REGION Network 60: STATUS - UNIT 01 - ST2
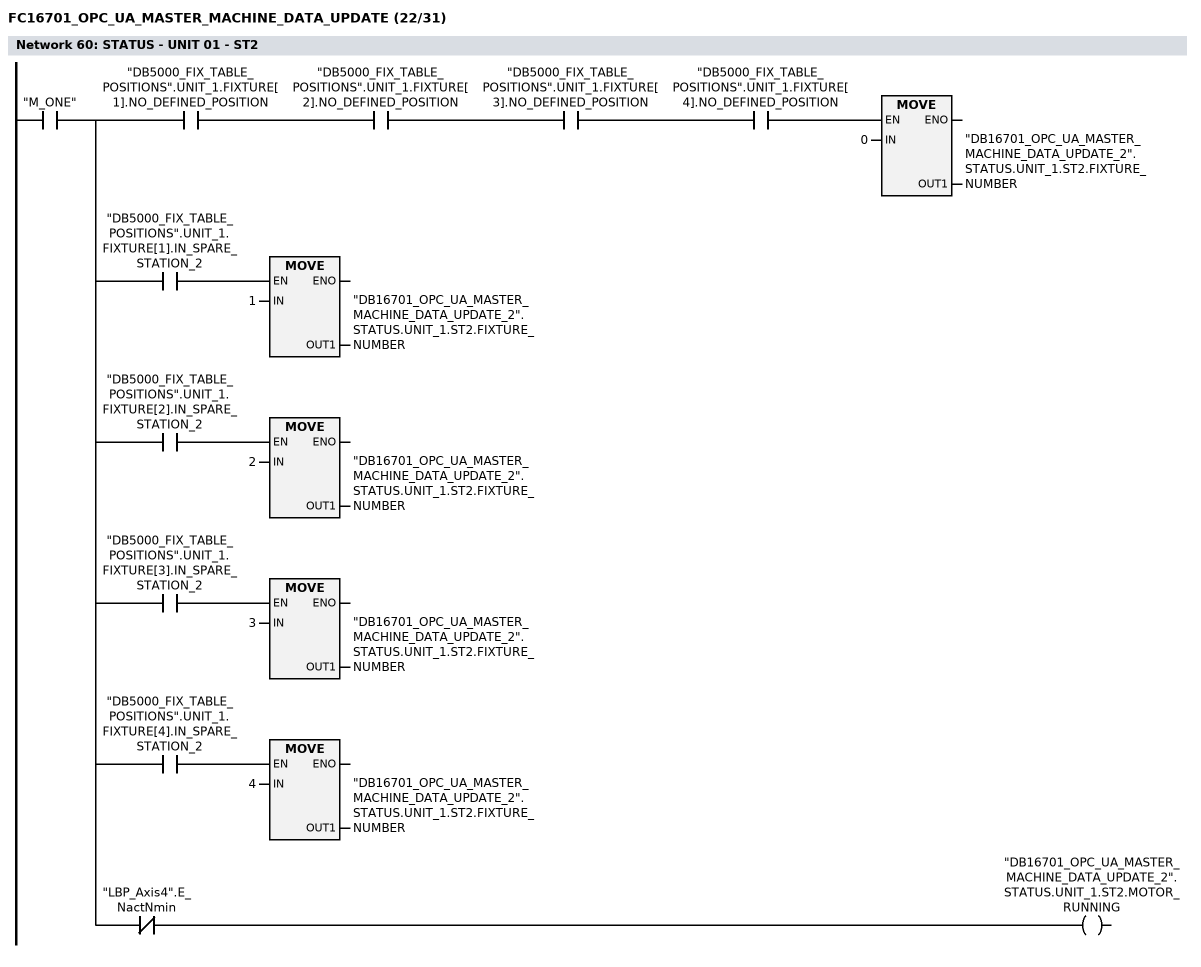
   RUNG wire#powerrail
      Contact( "M_ONE" )
      wire#w1
      Contact( "DB5000_FIX_TABLE_POSITIONS".UNIT_1.FIXTURE[1].NO_DEFINED_POSITION )
      Contact( "DB5000_FIX_TABLE_POSITIONS".UNIT_1.FIXTURE[2].NO_DEFINED_POSITION )
      Contact( "DB5000_FIX_TABLE_POSITIONS".UNIT_1.FIXTURE[3].NO_DEFINED_POSITION )
      Contact( "DB5000_FIX_TABLE_POSITIONS".UNIT_1.FIXTURE[4].NO_DEFINED_POSITION )
      Move(in := 0, out1 => "DB16701_OPC_UA_MASTER_MACHINE_DATA_UPDATE_2".STATUS.UNIT_1.ST2.FIXTURE_NUMBER)
   END_RUNG
   RUNG wire#w1
      Contact( "DB5000_FIX_TABLE_POSITIONS".UNIT_1.FIXTURE[1].IN_SPARE_STATION_2 )
      Move(in := 1, out1 => "DB16701_OPC_UA_MASTER_MACHINE_DATA_UPDATE_2".STATUS.UNIT_1.ST2.FIXTURE_NUMBER)
   END_RUNG
   RUNG wire#w1
      Contact( "DB5000_FIX_TABLE_POSITIONS".UNIT_1.FIXTURE[2].IN_SPARE_STATION_2 )
      Move(in := 2, out1 => "DB16701_OPC_UA_MASTER_MACHINE_DATA_UPDATE_2".STATUS.UNIT_1.ST2.FIXTURE_NUMBER)
   END_RUNG
   RUNG wire#w1
      Contact( "DB5000_FIX_TABLE_POSITIONS".UNIT_1.FIXTURE[3].IN_SPARE_STATION_2 )
      Move(in := 3, out1 => "DB16701_OPC_UA_MASTER_MACHINE_DATA_UPDATE_2".STATUS.UNIT_1.ST2.FIXTURE_NUMBER)
   END_RUNG
   RUNG wire#w1
      Contact( "DB5000_FIX_TABLE_POSITIONS".UNIT_1.FIXTURE[4].IN_SPARE_STATION_2 )
      Move(in := 4, out1 => "DB16701_OPC_UA_MASTER_MACHINE_DATA_UPDATE_2".STATUS.UNIT_1.ST2.FIXTURE_NUMBER)
   END_RUNG
   RUNG wire#w1
      I_Contact( "LBP_Axis4".E_NactNmin )
      Coil( "DB16701_OPC_UA_MASTER_MACHINE_DATA_UPDATE_2".STATUS.UNIT_1.ST2.MOTOR_RUNNING )
   END_RUNG
   // the same network as SCL:
   IF "M_ONE" AND "DB5000_FIX_TABLE_POSITIONS".UNIT_1.FIXTURE[1].NO_DEFINED_POSITION AND "DB5000_FIX_TABLE_POSITIONS".UNIT_1.FIXTURE[2].NO_DEFINED_POSITION AND "DB5000_FIX_TABLE_POSITIONS".UNIT_1.FIXTURE[3].NO_DEFINED_POSITION AND "DB5000_FIX_TABLE_POSITIONS".UNIT_1.FIXTURE[4].NO_DEFINED_POSITION THEN
       "DB16701_OPC_UA_MASTER_MACHINE_DATA_UPDATE_2".STATUS.UNIT_1.ST2.FIXTURE_NUMBER := 0;
   END_IF;
   IF "M_ONE" AND "DB5000_FIX_TABLE_POSITIONS".UNIT_1.FIXTURE[1].IN_SPARE_STATION_2 THEN
       "DB16701_OPC_UA_MASTER_MACHINE_DATA_UPDATE_2".STATUS.UNIT_1.ST2.FIXTURE_NUMBER := 1;
   END_IF;
   IF "M_ONE" AND "DB5000_FIX_TABLE_POSITIONS".UNIT_1.FIXTURE[2].IN_SPARE_STATION_2 THEN
       "DB16701_OPC_UA_MASTER_MACHINE_DATA_UPDATE_2".STATUS.UNIT_1.ST2.FIXTURE_NUMBER := 2;
   END_IF;
   IF "M_ONE" AND "DB5000_FIX_TABLE_POSITIONS".UNIT_1.FIXTURE[3].IN_SPARE_STATION_2 THEN
       "DB16701_OPC_UA_MASTER_MACHINE_DATA_UPDATE_2".STATUS.UNIT_1.ST2.FIXTURE_NUMBER := 3;
   END_IF;
   IF "M_ONE" AND "DB5000_FIX_TABLE_POSITIONS".UNIT_1.FIXTURE[4].IN_SPARE_STATION_2 THEN
       "DB16701_OPC_UA_MASTER_MACHINE_DATA_UPDATE_2".STATUS.UNIT_1.ST2.FIXTURE_NUMBER := 4;
   END_IF;
   "DB16701_OPC_UA_MASTER_MACHINE_DATA_UPDATE_2".STATUS.UNIT_1.ST2.MOTOR_RUNNING := "M_ONE" AND NOT "LBP_Axis4".E_NactNmin;
END_REGION

REGION Network 61: STATUS - UNIT 01 - ST3
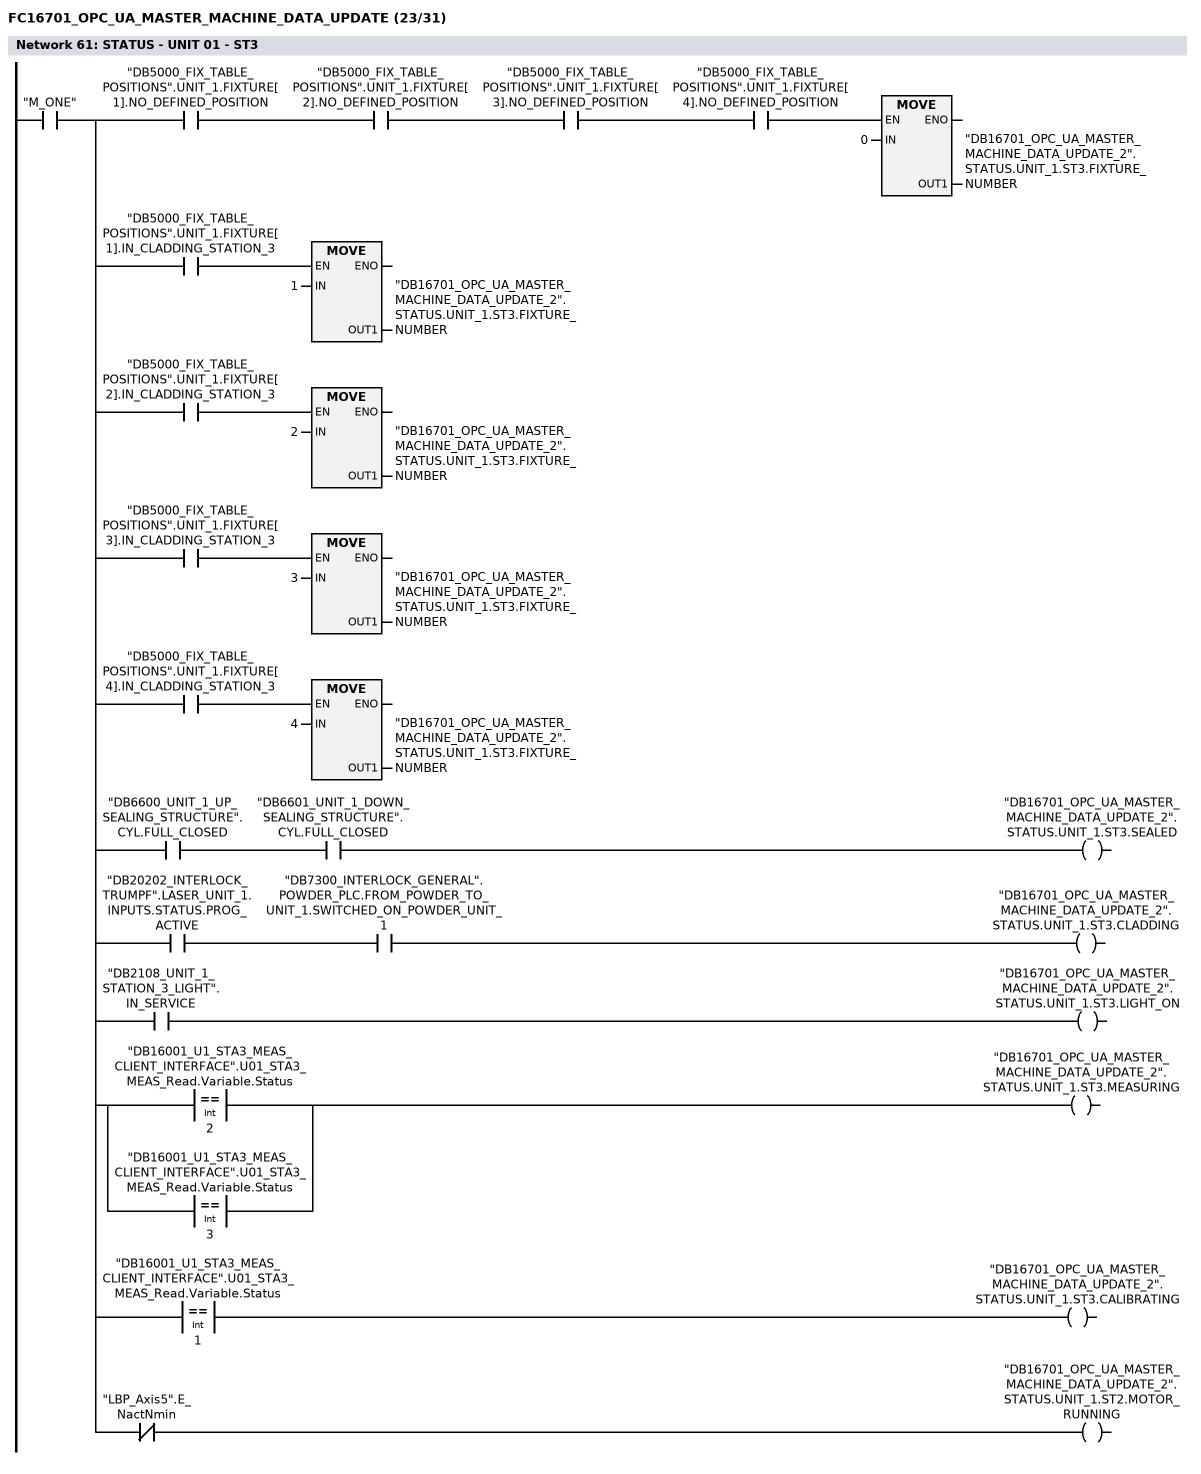
   RUNG wire#powerrail
      Contact( "M_ONE" )
      wire#w1
      Contact( "DB5000_FIX_TABLE_POSITIONS".UNIT_1.FIXTURE[1].NO_DEFINED_POSITION )
      Contact( "DB5000_FIX_TABLE_POSITIONS".UNIT_1.FIXTURE[2].NO_DEFINED_POSITION )
      Contact( "DB5000_FIX_TABLE_POSITIONS".UNIT_1.FIXTURE[3].NO_DEFINED_POSITION )
      Contact( "DB5000_FIX_TABLE_POSITIONS".UNIT_1.FIXTURE[4].NO_DEFINED_POSITION )
      Move(in := 0, out1 => "DB16701_OPC_UA_MASTER_MACHINE_DATA_UPDATE_2".STATUS.UNIT_1.ST3.FIXTURE_NUMBER)
   END_RUNG
   RUNG wire#w1
      Contact( "DB5000_FIX_TABLE_POSITIONS".UNIT_1.FIXTURE[1].IN_CLADDING_STATION_3 )
      Move(in := 1, out1 => "DB16701_OPC_UA_MASTER_MACHINE_DATA_UPDATE_2".STATUS.UNIT_1.ST3.FIXTURE_NUMBER)
   END_RUNG
   RUNG wire#w1
      Contact( "DB5000_FIX_TABLE_POSITIONS".UNIT_1.FIXTURE[2].IN_CLADDING_STATION_3 )
      Move(in := 2, out1 => "DB16701_OPC_UA_MASTER_MACHINE_DATA_UPDATE_2".STATUS.UNIT_1.ST3.FIXTURE_NUMBER)
   END_RUNG
   RUNG wire#w1
      Contact( "DB5000_FIX_TABLE_POSITIONS".UNIT_1.FIXTURE[3].IN_CLADDING_STATION_3 )
      Move(in := 3, out1 => "DB16701_OPC_UA_MASTER_MACHINE_DATA_UPDATE_2".STATUS.UNIT_1.ST3.FIXTURE_NUMBER)
   END_RUNG
   RUNG wire#w1
      Contact( "DB5000_FIX_TABLE_POSITIONS".UNIT_1.FIXTURE[4].IN_CLADDING_STATION_3 )
      Move(in := 4, out1 => "DB16701_OPC_UA_MASTER_MACHINE_DATA_UPDATE_2".STATUS.UNIT_1.ST3.FIXTURE_NUMBER)
   END_RUNG
   RUNG wire#w1
      Contact( "DB6600_UNIT_1_UP_SEALING_STRUCTURE".CYL.FULL_CLOSED )
      Contact( "DB6601_UNIT_1_DOWN_SEALING_STRUCTURE".CYL.FULL_CLOSED )
      Coil( "DB16701_OPC_UA_MASTER_MACHINE_DATA_UPDATE_2".STATUS.UNIT_1.ST3.SEALED )
   END_RUNG
   RUNG wire#w1
      Contact( "DB20202_INTERLOCK_TRUMPF".LASER_UNIT_1.INPUTS.STATUS.PROG_ACTIVE )
      Contact( "DB7300_INTERLOCK_GENERAL".POWDER_PLC.FROM_POWDER_TO_UNIT_1.SWITCHED_ON_POWDER_UNIT_1 )
      Coil( "DB16701_OPC_UA_MASTER_MACHINE_DATA_UPDATE_2".STATUS.UNIT_1.ST3.CLADDING )
   END_RUNG
   RUNG wire#w1
      Contact( "DB2108_UNIT_1_STATION_3_LIGHT".IN_SERVICE )
      Coil( "DB16701_OPC_UA_MASTER_MACHINE_DATA_UPDATE_2".STATUS.UNIT_1.ST3.LIGHT_ON )
   END_RUNG
   RUNG wire#w1
      { S7_Templates := "SrcType := Int" } EQ_Contact(in1 := "DB16001_U1_STA3_MEAS_CLIENT_INTERFACE".U01_STA3_MEAS_Read.Variable.Status, in2 := 2)
      wire#w2
      Coil( "DB16701_OPC_UA_MASTER_MACHINE_DATA_UPDATE_2".STATUS.UNIT_1.ST3.MEASURING )
   END_RUNG
   RUNG wire#w1
      { S7_Templates := "SrcType := Int" } EQ_Contact(in1 := "DB16001_U1_STA3_MEAS_CLIENT_INTERFACE".U01_STA3_MEAS_Read.Variable.Status, in2 := 3)
   END_RUNG wire#w2
   RUNG wire#w1
      { S7_Templates := "SrcType := Int" } EQ_Contact(in1 := "DB16001_U1_STA3_MEAS_CLIENT_INTERFACE".U01_STA3_MEAS_Read.Variable.Status, in2 := 1)
      Coil( "DB16701_OPC_UA_MASTER_MACHINE_DATA_UPDATE_2".STATUS.UNIT_1.ST3.CALIBRATING )
   END_RUNG
   RUNG wire#w1
      I_Contact( "LBP_Axis5".E_NactNmin )
      Coil( "DB16701_OPC_UA_MASTER_MACHINE_DATA_UPDATE_2".STATUS.UNIT_1.ST2.MOTOR_RUNNING )
   END_RUNG
   // the same network as SCL:
   IF "M_ONE" AND "DB5000_FIX_TABLE_POSITIONS".UNIT_1.FIXTURE[1].NO_DEFINED_POSITION AND "DB5000_FIX_TABLE_POSITIONS".UNIT_1.FIXTURE[2].NO_DEFINED_POSITION AND "DB5000_FIX_TABLE_POSITIONS".UNIT_1.FIXTURE[3].NO_DEFINED_POSITION AND "DB5000_FIX_TABLE_POSITIONS".UNIT_1.FIXTURE[4].NO_DEFINED_POSITION THEN
       "DB16701_OPC_UA_MASTER_MACHINE_DATA_UPDATE_2".STATUS.UNIT_1.ST3.FIXTURE_NUMBER := 0;
   END_IF;
   IF "M_ONE" AND "DB5000_FIX_TABLE_POSITIONS".UNIT_1.FIXTURE[1].IN_CLADDING_STATION_3 THEN
       "DB16701_OPC_UA_MASTER_MACHINE_DATA_UPDATE_2".STATUS.UNIT_1.ST3.FIXTURE_NUMBER := 1;
   END_IF;
   IF "M_ONE" AND "DB5000_FIX_TABLE_POSITIONS".UNIT_1.FIXTURE[2].IN_CLADDING_STATION_3 THEN
       "DB16701_OPC_UA_MASTER_MACHINE_DATA_UPDATE_2".STATUS.UNIT_1.ST3.FIXTURE_NUMBER := 2;
   END_IF;
   IF "M_ONE" AND "DB5000_FIX_TABLE_POSITIONS".UNIT_1.FIXTURE[3].IN_CLADDING_STATION_3 THEN
       "DB16701_OPC_UA_MASTER_MACHINE_DATA_UPDATE_2".STATUS.UNIT_1.ST3.FIXTURE_NUMBER := 3;
   END_IF;
   IF "M_ONE" AND "DB5000_FIX_TABLE_POSITIONS".UNIT_1.FIXTURE[4].IN_CLADDING_STATION_3 THEN
       "DB16701_OPC_UA_MASTER_MACHINE_DATA_UPDATE_2".STATUS.UNIT_1.ST3.FIXTURE_NUMBER := 4;
   END_IF;
   "DB16701_OPC_UA_MASTER_MACHINE_DATA_UPDATE_2".STATUS.UNIT_1.ST3.SEALED := "M_ONE" AND "DB6600_UNIT_1_UP_SEALING_STRUCTURE".CYL.FULL_CLOSED AND "DB6601_UNIT_1_DOWN_SEALING_STRUCTURE".CYL.FULL_CLOSED;
   "DB16701_OPC_UA_MASTER_MACHINE_DATA_UPDATE_2".STATUS.UNIT_1.ST3.CLADDING := "M_ONE" AND "DB20202_INTERLOCK_TRUMPF".LASER_UNIT_1.INPUTS.STATUS.PROG_ACTIVE AND "DB7300_INTERLOCK_GENERAL".POWDER_PLC.FROM_POWDER_TO_UNIT_1.SWITCHED_ON_POWDER_UNIT_1;
   "DB16701_OPC_UA_MASTER_MACHINE_DATA_UPDATE_2".STATUS.UNIT_1.ST3.LIGHT_ON := "M_ONE" AND "DB2108_UNIT_1_STATION_3_LIGHT".IN_SERVICE;
   "DB16701_OPC_UA_MASTER_MACHINE_DATA_UPDATE_2".STATUS.UNIT_1.ST3.MEASURING := "M_ONE" AND (("DB16001_U1_STA3_MEAS_CLIENT_INTERFACE".U01_STA3_MEAS_Read.Variable.Status = 2) OR ("DB16001_U1_STA3_MEAS_CLIENT_INTERFACE".U01_STA3_MEAS_Read.Variable.Status = 3));
   "DB16701_OPC_UA_MASTER_MACHINE_DATA_UPDATE_2".STATUS.UNIT_1.ST3.CALIBRATING := "M_ONE" AND ("DB16001_U1_STA3_MEAS_CLIENT_INTERFACE".U01_STA3_MEAS_Read.Variable.Status = 1);
   "DB16701_OPC_UA_MASTER_MACHINE_DATA_UPDATE_2".STATUS.UNIT_1.ST2.MOTOR_RUNNING := "M_ONE" AND NOT "LBP_Axis5".E_NactNmin;
END_REGION

REGION Network 62: STATUS - UNIT 01 - ST4
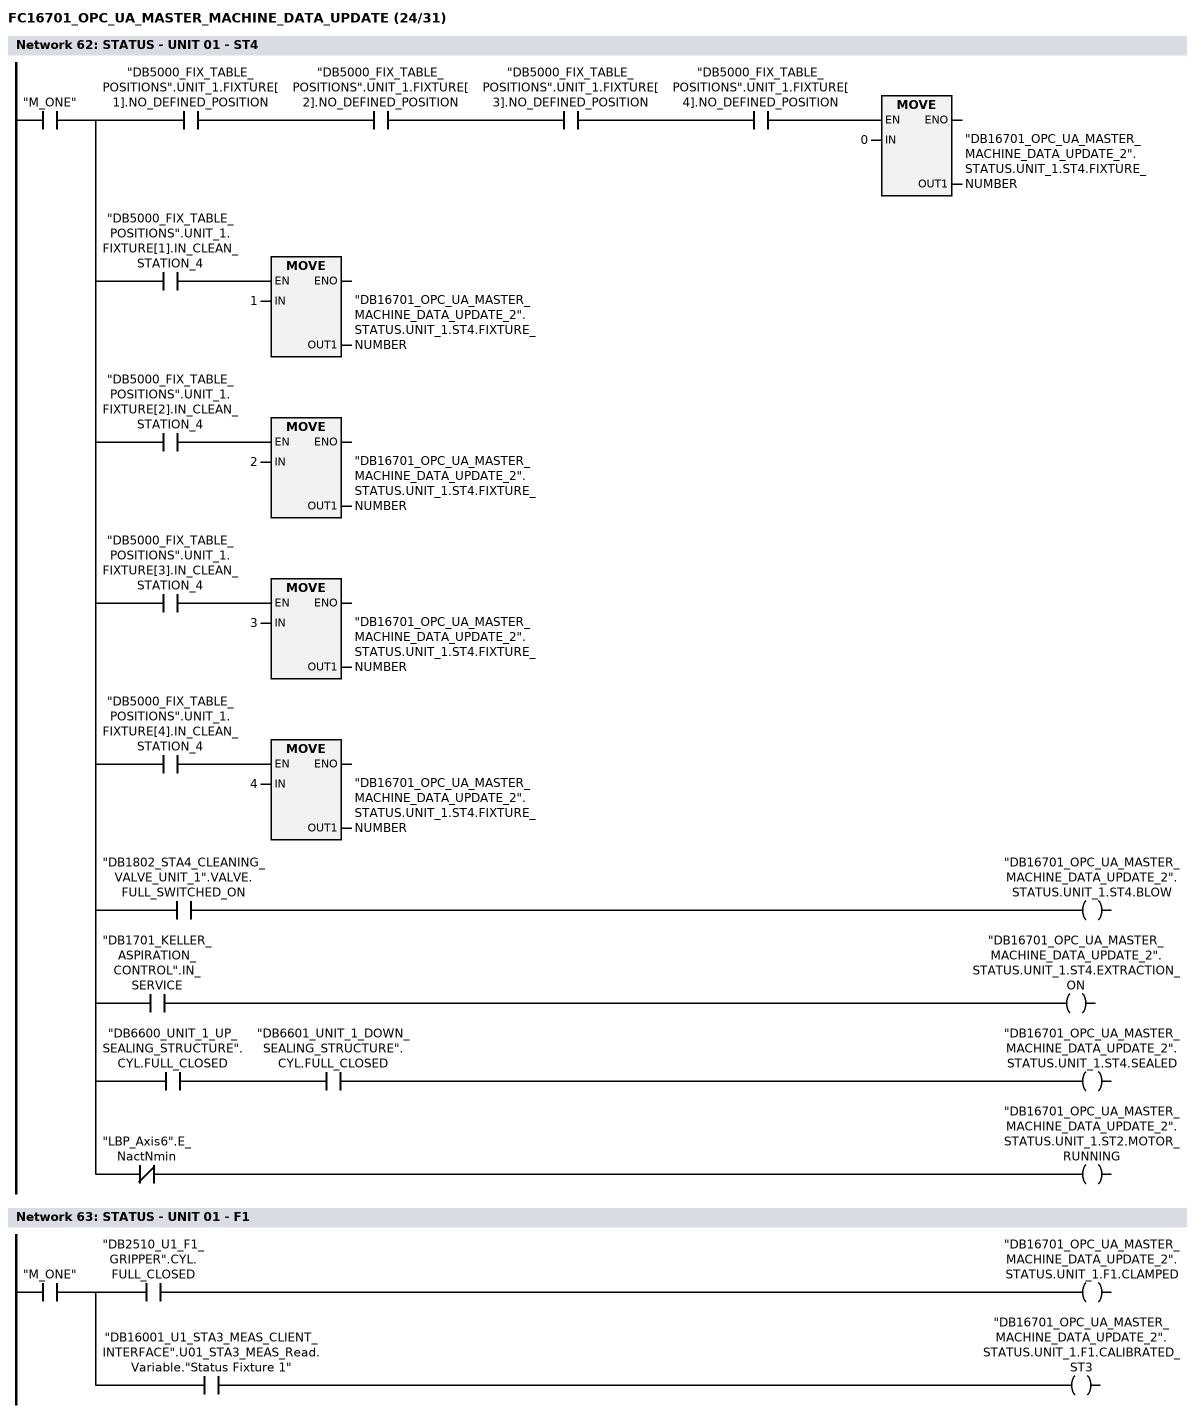
   RUNG wire#powerrail
      Contact( "M_ONE" )
      wire#w1
      Contact( "DB5000_FIX_TABLE_POSITIONS".UNIT_1.FIXTURE[1].NO_DEFINED_POSITION )
      Contact( "DB5000_FIX_TABLE_POSITIONS".UNIT_1.FIXTURE[2].NO_DEFINED_POSITION )
      Contact( "DB5000_FIX_TABLE_POSITIONS".UNIT_1.FIXTURE[3].NO_DEFINED_POSITION )
      Contact( "DB5000_FIX_TABLE_POSITIONS".UNIT_1.FIXTURE[4].NO_DEFINED_POSITION )
      Move(in := 0, out1 => "DB16701_OPC_UA_MASTER_MACHINE_DATA_UPDATE_2".STATUS.UNIT_1.ST4.FIXTURE_NUMBER)
   END_RUNG
   RUNG wire#w1
      Contact( "DB5000_FIX_TABLE_POSITIONS".UNIT_1.FIXTURE[1].IN_CLEAN_STATION_4 )
      Move(in := 1, out1 => "DB16701_OPC_UA_MASTER_MACHINE_DATA_UPDATE_2".STATUS.UNIT_1.ST4.FIXTURE_NUMBER)
   END_RUNG
   RUNG wire#w1
      Contact( "DB5000_FIX_TABLE_POSITIONS".UNIT_1.FIXTURE[2].IN_CLEAN_STATION_4 )
      Move(in := 2, out1 => "DB16701_OPC_UA_MASTER_MACHINE_DATA_UPDATE_2".STATUS.UNIT_1.ST4.FIXTURE_NUMBER)
   END_RUNG
   RUNG wire#w1
      Contact( "DB5000_FIX_TABLE_POSITIONS".UNIT_1.FIXTURE[3].IN_CLEAN_STATION_4 )
      Move(in := 3, out1 => "DB16701_OPC_UA_MASTER_MACHINE_DATA_UPDATE_2".STATUS.UNIT_1.ST4.FIXTURE_NUMBER)
   END_RUNG
   RUNG wire#w1
      Contact( "DB5000_FIX_TABLE_POSITIONS".UNIT_1.FIXTURE[4].IN_CLEAN_STATION_4 )
      Move(in := 4, out1 => "DB16701_OPC_UA_MASTER_MACHINE_DATA_UPDATE_2".STATUS.UNIT_1.ST4.FIXTURE_NUMBER)
   END_RUNG
   RUNG wire#w1
      Contact( "DB1802_STA4_CLEANING_VALVE_UNIT_1".VALVE.FULL_SWITCHED_ON )
      Coil( "DB16701_OPC_UA_MASTER_MACHINE_DATA_UPDATE_2".STATUS.UNIT_1.ST4.BLOW )
   END_RUNG
   RUNG wire#w1
      Contact( "DB1701_KELLER_ASPIRATION_CONTROL".IN_SERVICE )
      Coil( "DB16701_OPC_UA_MASTER_MACHINE_DATA_UPDATE_2".STATUS.UNIT_1.ST4.EXTRACTION_ON )
   END_RUNG
   RUNG wire#w1
      Contact( "DB6600_UNIT_1_UP_SEALING_STRUCTURE".CYL.FULL_CLOSED )
      Contact( "DB6601_UNIT_1_DOWN_SEALING_STRUCTURE".CYL.FULL_CLOSED )
      Coil( "DB16701_OPC_UA_MASTER_MACHINE_DATA_UPDATE_2".STATUS.UNIT_1.ST4.SEALED )
   END_RUNG
   RUNG wire#w1
      I_Contact( "LBP_Axis6".E_NactNmin )
      Coil( "DB16701_OPC_UA_MASTER_MACHINE_DATA_UPDATE_2".STATUS.UNIT_1.ST2.MOTOR_RUNNING )
   END_RUNG
   // the same network as SCL:
   IF "M_ONE" AND "DB5000_FIX_TABLE_POSITIONS".UNIT_1.FIXTURE[1].NO_DEFINED_POSITION AND "DB5000_FIX_TABLE_POSITIONS".UNIT_1.FIXTURE[2].NO_DEFINED_POSITION AND "DB5000_FIX_TABLE_POSITIONS".UNIT_1.FIXTURE[3].NO_DEFINED_POSITION AND "DB5000_FIX_TABLE_POSITIONS".UNIT_1.FIXTURE[4].NO_DEFINED_POSITION THEN
       "DB16701_OPC_UA_MASTER_MACHINE_DATA_UPDATE_2".STATUS.UNIT_1.ST4.FIXTURE_NUMBER := 0;
   END_IF;
   IF "M_ONE" AND "DB5000_FIX_TABLE_POSITIONS".UNIT_1.FIXTURE[1].IN_CLEAN_STATION_4 THEN
       "DB16701_OPC_UA_MASTER_MACHINE_DATA_UPDATE_2".STATUS.UNIT_1.ST4.FIXTURE_NUMBER := 1;
   END_IF;
   IF "M_ONE" AND "DB5000_FIX_TABLE_POSITIONS".UNIT_1.FIXTURE[2].IN_CLEAN_STATION_4 THEN
       "DB16701_OPC_UA_MASTER_MACHINE_DATA_UPDATE_2".STATUS.UNIT_1.ST4.FIXTURE_NUMBER := 2;
   END_IF;
   IF "M_ONE" AND "DB5000_FIX_TABLE_POSITIONS".UNIT_1.FIXTURE[3].IN_CLEAN_STATION_4 THEN
       "DB16701_OPC_UA_MASTER_MACHINE_DATA_UPDATE_2".STATUS.UNIT_1.ST4.FIXTURE_NUMBER := 3;
   END_IF;
   IF "M_ONE" AND "DB5000_FIX_TABLE_POSITIONS".UNIT_1.FIXTURE[4].IN_CLEAN_STATION_4 THEN
       "DB16701_OPC_UA_MASTER_MACHINE_DATA_UPDATE_2".STATUS.UNIT_1.ST4.FIXTURE_NUMBER := 4;
   END_IF;
   "DB16701_OPC_UA_MASTER_MACHINE_DATA_UPDATE_2".STATUS.UNIT_1.ST4.BLOW := "M_ONE" AND "DB1802_STA4_CLEANING_VALVE_UNIT_1".VALVE.FULL_SWITCHED_ON;
   "DB16701_OPC_UA_MASTER_MACHINE_DATA_UPDATE_2".STATUS.UNIT_1.ST4.EXTRACTION_ON := "M_ONE" AND "DB1701_KELLER_ASPIRATION_CONTROL".IN_SERVICE;
   "DB16701_OPC_UA_MASTER_MACHINE_DATA_UPDATE_2".STATUS.UNIT_1.ST4.SEALED := "M_ONE" AND "DB6600_UNIT_1_UP_SEALING_STRUCTURE".CYL.FULL_CLOSED AND "DB6601_UNIT_1_DOWN_SEALING_STRUCTURE".CYL.FULL_CLOSED;
   "DB16701_OPC_UA_MASTER_MACHINE_DATA_UPDATE_2".STATUS.UNIT_1.ST2.MOTOR_RUNNING := "M_ONE" AND NOT "LBP_Axis6".E_NactNmin;
END_REGION

REGION Network 63: STATUS - UNIT 01 - F1
   RUNG wire#powerrail
      Contact( "M_ONE" )
      wire#w1
      Contact( "DB2510_U1_F1_GRIPPER".CYL.FULL_CLOSED )
      Coil( "DB16701_OPC_UA_MASTER_MACHINE_DATA_UPDATE_2".STATUS.UNIT_1.F1.CLAMPED )
   END_RUNG
   RUNG wire#w1
      Contact( "DB16001_U1_STA3_MEAS_CLIENT_INTERFACE".U01_STA3_MEAS_Read.Variable."Status Fixture 1" )
      Coil( "DB16701_OPC_UA_MASTER_MACHINE_DATA_UPDATE_2".STATUS.UNIT_1.F1.CALIBRATED_ST3 )
   END_RUNG
   // the same network as SCL:
   "DB16701_OPC_UA_MASTER_MACHINE_DATA_UPDATE_2".STATUS.UNIT_1.F1.CLAMPED := "M_ONE" AND "DB2510_U1_F1_GRIPPER".CYL.FULL_CLOSED;
   "DB16701_OPC_UA_MASTER_MACHINE_DATA_UPDATE_2".STATUS.UNIT_1.F1.CALIBRATED_ST3 := "M_ONE" AND "DB16001_U1_STA3_MEAS_CLIENT_INTERFACE".U01_STA3_MEAS_Read.Variable."Status Fixture 1";
END_REGION

REGION Network 64: STATUS - UNIT 01 - F2
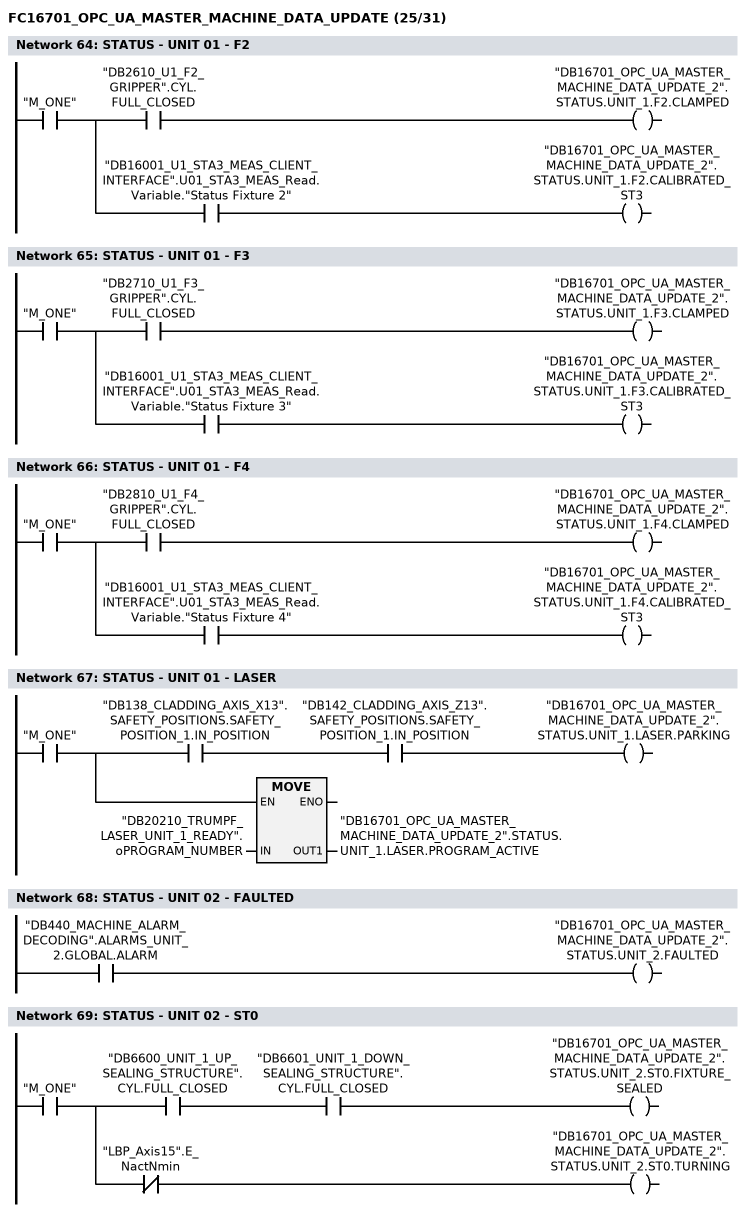
   RUNG wire#powerrail
      Contact( "M_ONE" )
      wire#w1
      Contact( "DB2610_U1_F2_GRIPPER".CYL.FULL_CLOSED )
      Coil( "DB16701_OPC_UA_MASTER_MACHINE_DATA_UPDATE_2".STATUS.UNIT_1.F2.CLAMPED )
   END_RUNG
   RUNG wire#w1
      Contact( "DB16001_U1_STA3_MEAS_CLIENT_INTERFACE".U01_STA3_MEAS_Read.Variable."Status Fixture 2" )
      Coil( "DB16701_OPC_UA_MASTER_MACHINE_DATA_UPDATE_2".STATUS.UNIT_1.F2.CALIBRATED_ST3 )
   END_RUNG
   // the same network as SCL:
   "DB16701_OPC_UA_MASTER_MACHINE_DATA_UPDATE_2".STATUS.UNIT_1.F2.CLAMPED := "M_ONE" AND "DB2610_U1_F2_GRIPPER".CYL.FULL_CLOSED;
   "DB16701_OPC_UA_MASTER_MACHINE_DATA_UPDATE_2".STATUS.UNIT_1.F2.CALIBRATED_ST3 := "M_ONE" AND "DB16001_U1_STA3_MEAS_CLIENT_INTERFACE".U01_STA3_MEAS_Read.Variable."Status Fixture 2";
END_REGION

REGION Network 65: STATUS - UNIT 01 - F3
   RUNG wire#powerrail
      Contact( "M_ONE" )
      wire#w1
      Contact( "DB2710_U1_F3_GRIPPER".CYL.FULL_CLOSED )
      Coil( "DB16701_OPC_UA_MASTER_MACHINE_DATA_UPDATE_2".STATUS.UNIT_1.F3.CLAMPED )
   END_RUNG
   RUNG wire#w1
      Contact( "DB16001_U1_STA3_MEAS_CLIENT_INTERFACE".U01_STA3_MEAS_Read.Variable."Status Fixture 3" )
      Coil( "DB16701_OPC_UA_MASTER_MACHINE_DATA_UPDATE_2".STATUS.UNIT_1.F3.CALIBRATED_ST3 )
   END_RUNG
   // the same network as SCL:
   "DB16701_OPC_UA_MASTER_MACHINE_DATA_UPDATE_2".STATUS.UNIT_1.F3.CLAMPED := "M_ONE" AND "DB2710_U1_F3_GRIPPER".CYL.FULL_CLOSED;
   "DB16701_OPC_UA_MASTER_MACHINE_DATA_UPDATE_2".STATUS.UNIT_1.F3.CALIBRATED_ST3 := "M_ONE" AND "DB16001_U1_STA3_MEAS_CLIENT_INTERFACE".U01_STA3_MEAS_Read.Variable."Status Fixture 3";
END_REGION

REGION Network 66: STATUS - UNIT 01 - F4
   RUNG wire#powerrail
      Contact( "M_ONE" )
      wire#w1
      Contact( "DB2810_U1_F4_GRIPPER".CYL.FULL_CLOSED )
      Coil( "DB16701_OPC_UA_MASTER_MACHINE_DATA_UPDATE_2".STATUS.UNIT_1.F4.CLAMPED )
   END_RUNG
   RUNG wire#w1
      Contact( "DB16001_U1_STA3_MEAS_CLIENT_INTERFACE".U01_STA3_MEAS_Read.Variable."Status Fixture 4" )
      Coil( "DB16701_OPC_UA_MASTER_MACHINE_DATA_UPDATE_2".STATUS.UNIT_1.F4.CALIBRATED_ST3 )
   END_RUNG
   // the same network as SCL:
   "DB16701_OPC_UA_MASTER_MACHINE_DATA_UPDATE_2".STATUS.UNIT_1.F4.CLAMPED := "M_ONE" AND "DB2810_U1_F4_GRIPPER".CYL.FULL_CLOSED;
   "DB16701_OPC_UA_MASTER_MACHINE_DATA_UPDATE_2".STATUS.UNIT_1.F4.CALIBRATED_ST3 := "M_ONE" AND "DB16001_U1_STA3_MEAS_CLIENT_INTERFACE".U01_STA3_MEAS_Read.Variable."Status Fixture 4";
END_REGION

REGION Network 67: STATUS - UNIT 01 - LASER
   RUNG wire#powerrail
      Contact( "M_ONE" )
      wire#w1
      Contact( "DB138_CLADDING_AXIS_X13".SAFETY_POSITIONS.SAFETY_POSITION_1.IN_POSITION )
      Contact( "DB142_CLADDING_AXIS_Z13".SAFETY_POSITIONS.SAFETY_POSITION_1.IN_POSITION )
      Coil( "DB16701_OPC_UA_MASTER_MACHINE_DATA_UPDATE_2".STATUS.UNIT_1.LASER.PARKING )
   END_RUNG
   RUNG wire#w1
      Move(in := "DB20210_TRUMPF_LASER_UNIT_1_READY".oPROGRAM_NUMBER, out1 => "DB16701_OPC_UA_MASTER_MACHINE_DATA_UPDATE_2".STATUS.UNIT_1.LASER.PROGRAM_ACTIVE)
   END_RUNG
   // the same network as SCL:
   "DB16701_OPC_UA_MASTER_MACHINE_DATA_UPDATE_2".STATUS.UNIT_1.LASER.PARKING := "M_ONE" AND "DB138_CLADDING_AXIS_X13".SAFETY_POSITIONS.SAFETY_POSITION_1.IN_POSITION AND "DB142_CLADDING_AXIS_Z13".SAFETY_POSITIONS.SAFETY_POSITION_1.IN_POSITION;
   IF "M_ONE" THEN
       "DB16701_OPC_UA_MASTER_MACHINE_DATA_UPDATE_2".STATUS.UNIT_1.LASER.PROGRAM_ACTIVE := "DB20210_TRUMPF_LASER_UNIT_1_READY".oPROGRAM_NUMBER;
   END_IF;
END_REGION

REGION Network 68: STATUS - UNIT 02 - FAULTED
   RUNG wire#powerrail
      Contact( "DB440_MACHINE_ALARM_DECODING".ALARMS_UNIT_2.GLOBAL.ALARM )
      Coil( "DB16701_OPC_UA_MASTER_MACHINE_DATA_UPDATE_2".STATUS.UNIT_2.FAULTED )
   END_RUNG
   // the same network as SCL:
   "DB16701_OPC_UA_MASTER_MACHINE_DATA_UPDATE_2".STATUS.UNIT_2.FAULTED := "DB440_MACHINE_ALARM_DECODING".ALARMS_UNIT_2.GLOBAL.ALARM;
END_REGION

REGION Network 69: STATUS - UNIT 02 - ST0
   RUNG wire#powerrail
      Contact( "M_ONE" )
      wire#w1
      Contact( "DB6600_UNIT_1_UP_SEALING_STRUCTURE".CYL.FULL_CLOSED )
      Contact( "DB6601_UNIT_1_DOWN_SEALING_STRUCTURE".CYL.FULL_CLOSED )
      Coil( "DB16701_OPC_UA_MASTER_MACHINE_DATA_UPDATE_2".STATUS.UNIT_2.ST0.FIXTURE_SEALED )
   END_RUNG
   RUNG wire#w1
      I_Contact( "LBP_Axis15".E_NactNmin )
      Coil( "DB16701_OPC_UA_MASTER_MACHINE_DATA_UPDATE_2".STATUS.UNIT_2.ST0.TURNING )
   END_RUNG
   // the same network as SCL:
   "DB16701_OPC_UA_MASTER_MACHINE_DATA_UPDATE_2".STATUS.UNIT_2.ST0.FIXTURE_SEALED := "M_ONE" AND "DB6600_UNIT_1_UP_SEALING_STRUCTURE".CYL.FULL_CLOSED AND "DB6601_UNIT_1_DOWN_SEALING_STRUCTURE".CYL.FULL_CLOSED;
   "DB16701_OPC_UA_MASTER_MACHINE_DATA_UPDATE_2".STATUS.UNIT_2.ST0.TURNING := "M_ONE" AND NOT "LBP_Axis15".E_NactNmin;
END_REGION

REGION Network 70: STATUS - UNIT 02 - ST1
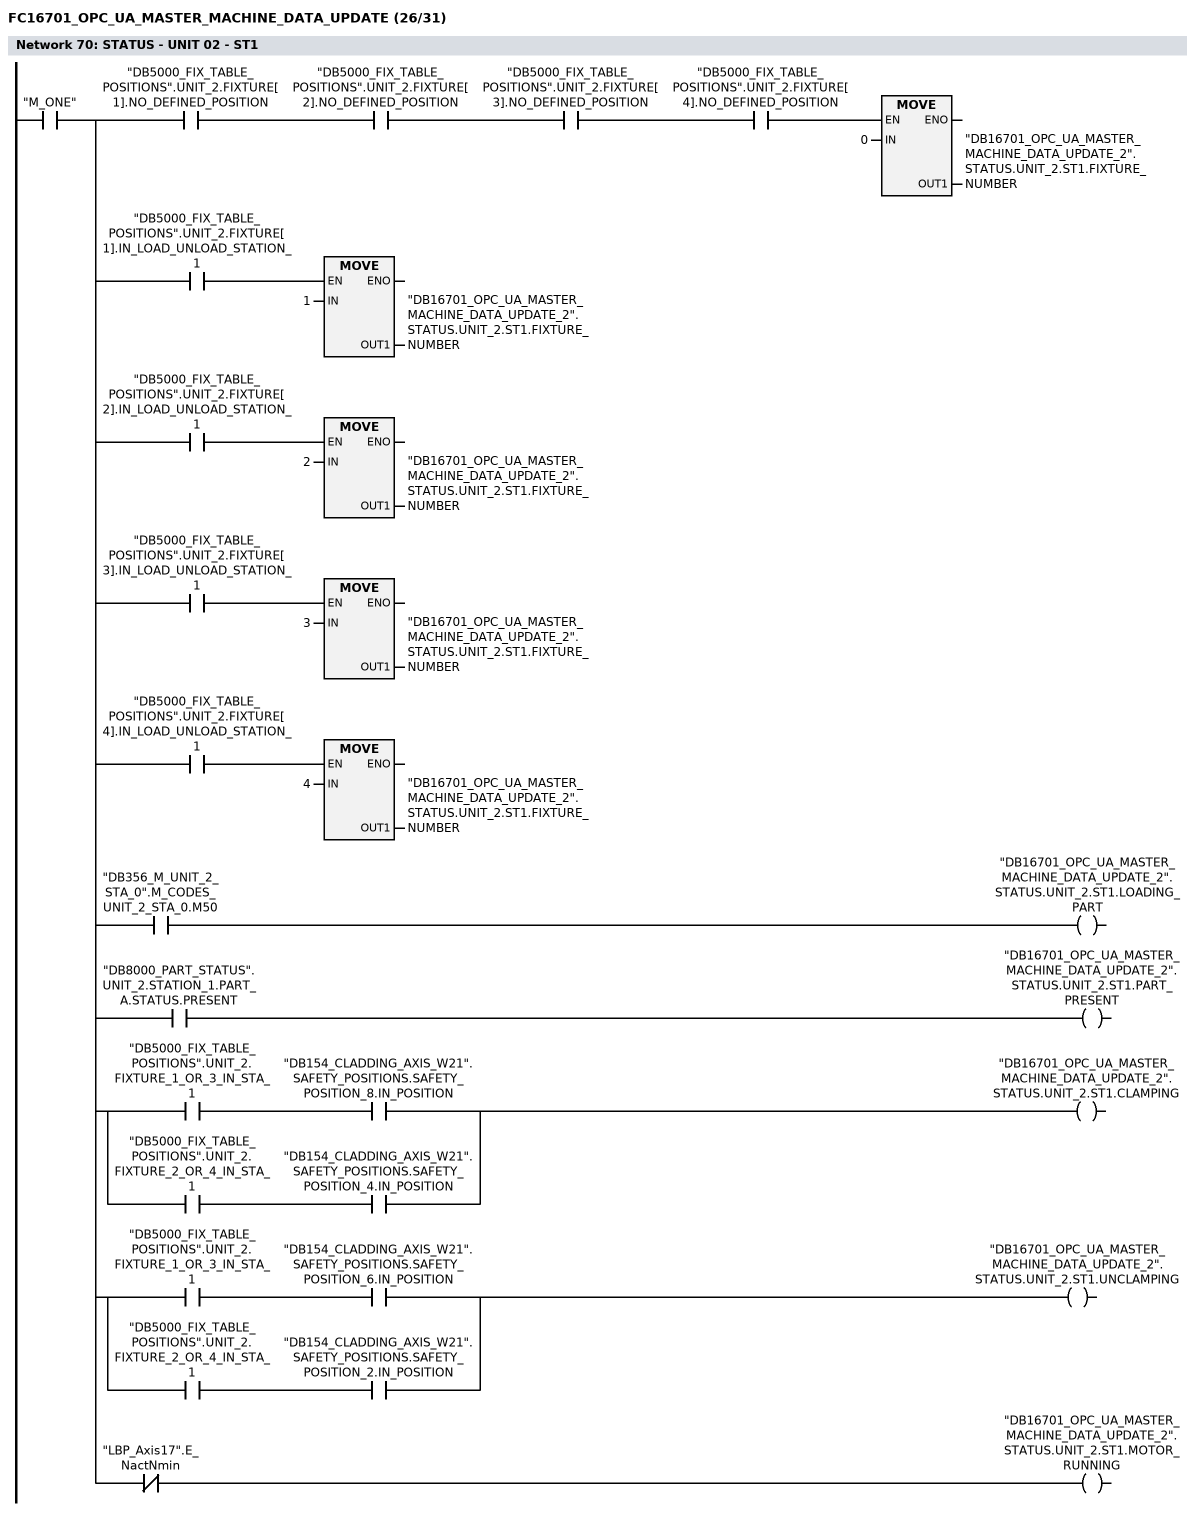
   RUNG wire#powerrail
      Contact( "M_ONE" )
      wire#w1
      Contact( "DB5000_FIX_TABLE_POSITIONS".UNIT_2.FIXTURE[1].NO_DEFINED_POSITION )
      Contact( "DB5000_FIX_TABLE_POSITIONS".UNIT_2.FIXTURE[2].NO_DEFINED_POSITION )
      Contact( "DB5000_FIX_TABLE_POSITIONS".UNIT_2.FIXTURE[3].NO_DEFINED_POSITION )
      Contact( "DB5000_FIX_TABLE_POSITIONS".UNIT_2.FIXTURE[4].NO_DEFINED_POSITION )
      Move(in := 0, out1 => "DB16701_OPC_UA_MASTER_MACHINE_DATA_UPDATE_2".STATUS.UNIT_2.ST1.FIXTURE_NUMBER)
   END_RUNG
   RUNG wire#w1
      Contact( "DB5000_FIX_TABLE_POSITIONS".UNIT_2.FIXTURE[1].IN_LOAD_UNLOAD_STATION_1 )
      Move(in := 1, out1 => "DB16701_OPC_UA_MASTER_MACHINE_DATA_UPDATE_2".STATUS.UNIT_2.ST1.FIXTURE_NUMBER)
   END_RUNG
   RUNG wire#w1
      Contact( "DB5000_FIX_TABLE_POSITIONS".UNIT_2.FIXTURE[2].IN_LOAD_UNLOAD_STATION_1 )
      Move(in := 2, out1 => "DB16701_OPC_UA_MASTER_MACHINE_DATA_UPDATE_2".STATUS.UNIT_2.ST1.FIXTURE_NUMBER)
   END_RUNG
   RUNG wire#w1
      Contact( "DB5000_FIX_TABLE_POSITIONS".UNIT_2.FIXTURE[3].IN_LOAD_UNLOAD_STATION_1 )
      Move(in := 3, out1 => "DB16701_OPC_UA_MASTER_MACHINE_DATA_UPDATE_2".STATUS.UNIT_2.ST1.FIXTURE_NUMBER)
   END_RUNG
   RUNG wire#w1
      Contact( "DB5000_FIX_TABLE_POSITIONS".UNIT_2.FIXTURE[4].IN_LOAD_UNLOAD_STATION_1 )
      Move(in := 4, out1 => "DB16701_OPC_UA_MASTER_MACHINE_DATA_UPDATE_2".STATUS.UNIT_2.ST1.FIXTURE_NUMBER)
   END_RUNG
   RUNG wire#w1
      Contact( "DB356_M_UNIT_2_STA_0".M_CODES_UNIT_2_STA_0.M50 )
      Coil( "DB16701_OPC_UA_MASTER_MACHINE_DATA_UPDATE_2".STATUS.UNIT_2.ST1.LOADING_PART )
   END_RUNG
   RUNG wire#w1
      Contact( "DB8000_PART_STATUS".UNIT_2.STATION_1.PART_A.STATUS.PRESENT )
      Coil( "DB16701_OPC_UA_MASTER_MACHINE_DATA_UPDATE_2".STATUS.UNIT_2.ST1.PART_PRESENT )
   END_RUNG
   RUNG wire#w1
      Contact( "DB5000_FIX_TABLE_POSITIONS".UNIT_2.FIXTURE_1_OR_3_IN_STA_1 )
      Contact( "DB154_CLADDING_AXIS_W21".SAFETY_POSITIONS.SAFETY_POSITION_8.IN_POSITION )
      wire#w2
      Coil( "DB16701_OPC_UA_MASTER_MACHINE_DATA_UPDATE_2".STATUS.UNIT_2.ST1.CLAMPING )
   END_RUNG
   RUNG wire#w1
      Contact( "DB5000_FIX_TABLE_POSITIONS".UNIT_2.FIXTURE_2_OR_4_IN_STA_1 )
      Contact( "DB154_CLADDING_AXIS_W21".SAFETY_POSITIONS.SAFETY_POSITION_4.IN_POSITION )
   END_RUNG wire#w2
   RUNG wire#w1
      Contact( "DB5000_FIX_TABLE_POSITIONS".UNIT_2.FIXTURE_1_OR_3_IN_STA_1 )
      Contact( "DB154_CLADDING_AXIS_W21".SAFETY_POSITIONS.SAFETY_POSITION_6.IN_POSITION )
      wire#w3
      Coil( "DB16701_OPC_UA_MASTER_MACHINE_DATA_UPDATE_2".STATUS.UNIT_2.ST1.UNCLAMPING )
   END_RUNG
   RUNG wire#w1
      Contact( "DB5000_FIX_TABLE_POSITIONS".UNIT_2.FIXTURE_2_OR_4_IN_STA_1 )
      Contact( "DB154_CLADDING_AXIS_W21".SAFETY_POSITIONS.SAFETY_POSITION_2.IN_POSITION )
   END_RUNG wire#w3
   RUNG wire#w1
      I_Contact( "LBP_Axis17".E_NactNmin )
      Coil( "DB16701_OPC_UA_MASTER_MACHINE_DATA_UPDATE_2".STATUS.UNIT_2.ST1.MOTOR_RUNNING )
   END_RUNG
   // the same network as SCL:
   IF "M_ONE" AND "DB5000_FIX_TABLE_POSITIONS".UNIT_2.FIXTURE[1].NO_DEFINED_POSITION AND "DB5000_FIX_TABLE_POSITIONS".UNIT_2.FIXTURE[2].NO_DEFINED_POSITION AND "DB5000_FIX_TABLE_POSITIONS".UNIT_2.FIXTURE[3].NO_DEFINED_POSITION AND "DB5000_FIX_TABLE_POSITIONS".UNIT_2.FIXTURE[4].NO_DEFINED_POSITION THEN
       "DB16701_OPC_UA_MASTER_MACHINE_DATA_UPDATE_2".STATUS.UNIT_2.ST1.FIXTURE_NUMBER := 0;
   END_IF;
   IF "M_ONE" AND "DB5000_FIX_TABLE_POSITIONS".UNIT_2.FIXTURE[1].IN_LOAD_UNLOAD_STATION_1 THEN
       "DB16701_OPC_UA_MASTER_MACHINE_DATA_UPDATE_2".STATUS.UNIT_2.ST1.FIXTURE_NUMBER := 1;
   END_IF;
   IF "M_ONE" AND "DB5000_FIX_TABLE_POSITIONS".UNIT_2.FIXTURE[2].IN_LOAD_UNLOAD_STATION_1 THEN
       "DB16701_OPC_UA_MASTER_MACHINE_DATA_UPDATE_2".STATUS.UNIT_2.ST1.FIXTURE_NUMBER := 2;
   END_IF;
   IF "M_ONE" AND "DB5000_FIX_TABLE_POSITIONS".UNIT_2.FIXTURE[3].IN_LOAD_UNLOAD_STATION_1 THEN
       "DB16701_OPC_UA_MASTER_MACHINE_DATA_UPDATE_2".STATUS.UNIT_2.ST1.FIXTURE_NUMBER := 3;
   END_IF;
   IF "M_ONE" AND "DB5000_FIX_TABLE_POSITIONS".UNIT_2.FIXTURE[4].IN_LOAD_UNLOAD_STATION_1 THEN
       "DB16701_OPC_UA_MASTER_MACHINE_DATA_UPDATE_2".STATUS.UNIT_2.ST1.FIXTURE_NUMBER := 4;
   END_IF;
   "DB16701_OPC_UA_MASTER_MACHINE_DATA_UPDATE_2".STATUS.UNIT_2.ST1.LOADING_PART := "M_ONE" AND "DB356_M_UNIT_2_STA_0".M_CODES_UNIT_2_STA_0.M50;
   "DB16701_OPC_UA_MASTER_MACHINE_DATA_UPDATE_2".STATUS.UNIT_2.ST1.PART_PRESENT := "M_ONE" AND "DB8000_PART_STATUS".UNIT_2.STATION_1.PART_A.STATUS.PRESENT;
   "DB16701_OPC_UA_MASTER_MACHINE_DATA_UPDATE_2".STATUS.UNIT_2.ST1.CLAMPING := "M_ONE" AND (("DB5000_FIX_TABLE_POSITIONS".UNIT_2.FIXTURE_1_OR_3_IN_STA_1 AND "DB154_CLADDING_AXIS_W21".SAFETY_POSITIONS.SAFETY_POSITION_8.IN_POSITION) OR ("DB5000_FIX_TABLE_POSITIONS".UNIT_2.FIXTURE_2_OR_4_IN_STA_1 AND "DB154_CLADDING_AXIS_W21".SAFETY_POSITIONS.SAFETY_POSITION_4.IN_POSITION));
   "DB16701_OPC_UA_MASTER_MACHINE_DATA_UPDATE_2".STATUS.UNIT_2.ST1.UNCLAMPING := "M_ONE" AND (("DB5000_FIX_TABLE_POSITIONS".UNIT_2.FIXTURE_1_OR_3_IN_STA_1 AND "DB154_CLADDING_AXIS_W21".SAFETY_POSITIONS.SAFETY_POSITION_6.IN_POSITION) OR ("DB5000_FIX_TABLE_POSITIONS".UNIT_2.FIXTURE_2_OR_4_IN_STA_1 AND "DB154_CLADDING_AXIS_W21".SAFETY_POSITIONS.SAFETY_POSITION_2.IN_POSITION));
   "DB16701_OPC_UA_MASTER_MACHINE_DATA_UPDATE_2".STATUS.UNIT_2.ST1.MOTOR_RUNNING := "M_ONE" AND NOT "LBP_Axis17".E_NactNmin;
END_REGION

REGION Network 71: STATUS - UNIT 02 - ST2
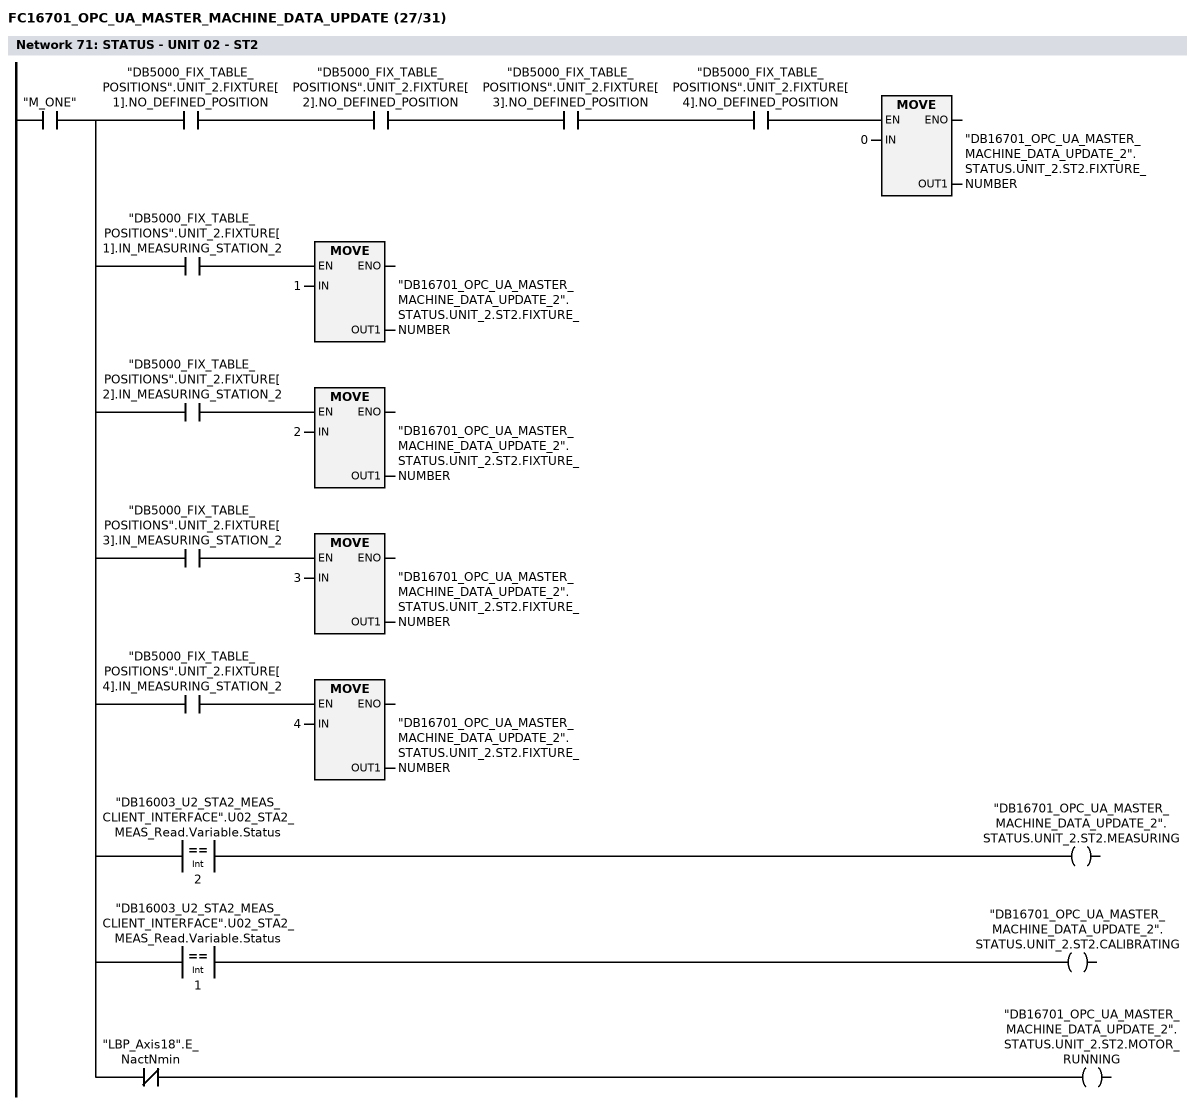
   RUNG wire#powerrail
      Contact( "M_ONE" )
      wire#w1
      Contact( "DB5000_FIX_TABLE_POSITIONS".UNIT_2.FIXTURE[1].NO_DEFINED_POSITION )
      Contact( "DB5000_FIX_TABLE_POSITIONS".UNIT_2.FIXTURE[2].NO_DEFINED_POSITION )
      Contact( "DB5000_FIX_TABLE_POSITIONS".UNIT_2.FIXTURE[3].NO_DEFINED_POSITION )
      Contact( "DB5000_FIX_TABLE_POSITIONS".UNIT_2.FIXTURE[4].NO_DEFINED_POSITION )
      Move(in := 0, out1 => "DB16701_OPC_UA_MASTER_MACHINE_DATA_UPDATE_2".STATUS.UNIT_2.ST2.FIXTURE_NUMBER)
   END_RUNG
   RUNG wire#w1
      Contact( "DB5000_FIX_TABLE_POSITIONS".UNIT_2.FIXTURE[1].IN_MEASURING_STATION_2 )
      Move(in := 1, out1 => "DB16701_OPC_UA_MASTER_MACHINE_DATA_UPDATE_2".STATUS.UNIT_2.ST2.FIXTURE_NUMBER)
   END_RUNG
   RUNG wire#w1
      Contact( "DB5000_FIX_TABLE_POSITIONS".UNIT_2.FIXTURE[2].IN_MEASURING_STATION_2 )
      Move(in := 2, out1 => "DB16701_OPC_UA_MASTER_MACHINE_DATA_UPDATE_2".STATUS.UNIT_2.ST2.FIXTURE_NUMBER)
   END_RUNG
   RUNG wire#w1
      Contact( "DB5000_FIX_TABLE_POSITIONS".UNIT_2.FIXTURE[3].IN_MEASURING_STATION_2 )
      Move(in := 3, out1 => "DB16701_OPC_UA_MASTER_MACHINE_DATA_UPDATE_2".STATUS.UNIT_2.ST2.FIXTURE_NUMBER)
   END_RUNG
   RUNG wire#w1
      Contact( "DB5000_FIX_TABLE_POSITIONS".UNIT_2.FIXTURE[4].IN_MEASURING_STATION_2 )
      Move(in := 4, out1 => "DB16701_OPC_UA_MASTER_MACHINE_DATA_UPDATE_2".STATUS.UNIT_2.ST2.FIXTURE_NUMBER)
   END_RUNG
   RUNG wire#w1
      { S7_Templates := "SrcType := Int" } EQ_Contact(in1 := "DB16003_U2_STA2_MEAS_CLIENT_INTERFACE".U02_STA2_MEAS_Read.Variable.Status, in2 := 2)
      Coil( "DB16701_OPC_UA_MASTER_MACHINE_DATA_UPDATE_2".STATUS.UNIT_2.ST2.MEASURING )
   END_RUNG
   RUNG wire#w1
      { S7_Templates := "SrcType := Int" } EQ_Contact(in1 := "DB16003_U2_STA2_MEAS_CLIENT_INTERFACE".U02_STA2_MEAS_Read.Variable.Status, in2 := 1)
      Coil( "DB16701_OPC_UA_MASTER_MACHINE_DATA_UPDATE_2".STATUS.UNIT_2.ST2.CALIBRATING )
   END_RUNG
   RUNG wire#w1
      I_Contact( "LBP_Axis18".E_NactNmin )
      Coil( "DB16701_OPC_UA_MASTER_MACHINE_DATA_UPDATE_2".STATUS.UNIT_2.ST2.MOTOR_RUNNING )
   END_RUNG
   // the same network as SCL:
   IF "M_ONE" AND "DB5000_FIX_TABLE_POSITIONS".UNIT_2.FIXTURE[1].NO_DEFINED_POSITION AND "DB5000_FIX_TABLE_POSITIONS".UNIT_2.FIXTURE[2].NO_DEFINED_POSITION AND "DB5000_FIX_TABLE_POSITIONS".UNIT_2.FIXTURE[3].NO_DEFINED_POSITION AND "DB5000_FIX_TABLE_POSITIONS".UNIT_2.FIXTURE[4].NO_DEFINED_POSITION THEN
       "DB16701_OPC_UA_MASTER_MACHINE_DATA_UPDATE_2".STATUS.UNIT_2.ST2.FIXTURE_NUMBER := 0;
   END_IF;
   IF "M_ONE" AND "DB5000_FIX_TABLE_POSITIONS".UNIT_2.FIXTURE[1].IN_MEASURING_STATION_2 THEN
       "DB16701_OPC_UA_MASTER_MACHINE_DATA_UPDATE_2".STATUS.UNIT_2.ST2.FIXTURE_NUMBER := 1;
   END_IF;
   IF "M_ONE" AND "DB5000_FIX_TABLE_POSITIONS".UNIT_2.FIXTURE[2].IN_MEASURING_STATION_2 THEN
       "DB16701_OPC_UA_MASTER_MACHINE_DATA_UPDATE_2".STATUS.UNIT_2.ST2.FIXTURE_NUMBER := 2;
   END_IF;
   IF "M_ONE" AND "DB5000_FIX_TABLE_POSITIONS".UNIT_2.FIXTURE[3].IN_MEASURING_STATION_2 THEN
       "DB16701_OPC_UA_MASTER_MACHINE_DATA_UPDATE_2".STATUS.UNIT_2.ST2.FIXTURE_NUMBER := 3;
   END_IF;
   IF "M_ONE" AND "DB5000_FIX_TABLE_POSITIONS".UNIT_2.FIXTURE[4].IN_MEASURING_STATION_2 THEN
       "DB16701_OPC_UA_MASTER_MACHINE_DATA_UPDATE_2".STATUS.UNIT_2.ST2.FIXTURE_NUMBER := 4;
   END_IF;
   "DB16701_OPC_UA_MASTER_MACHINE_DATA_UPDATE_2".STATUS.UNIT_2.ST2.MEASURING := "M_ONE" AND ("DB16003_U2_STA2_MEAS_CLIENT_INTERFACE".U02_STA2_MEAS_Read.Variable.Status = 2);
   "DB16701_OPC_UA_MASTER_MACHINE_DATA_UPDATE_2".STATUS.UNIT_2.ST2.CALIBRATING := "M_ONE" AND ("DB16003_U2_STA2_MEAS_CLIENT_INTERFACE".U02_STA2_MEAS_Read.Variable.Status = 1);
   "DB16701_OPC_UA_MASTER_MACHINE_DATA_UPDATE_2".STATUS.UNIT_2.ST2.MOTOR_RUNNING := "M_ONE" AND NOT "LBP_Axis18".E_NactNmin;
END_REGION

REGION Network 72: STATUS - UNIT 02 - ST3
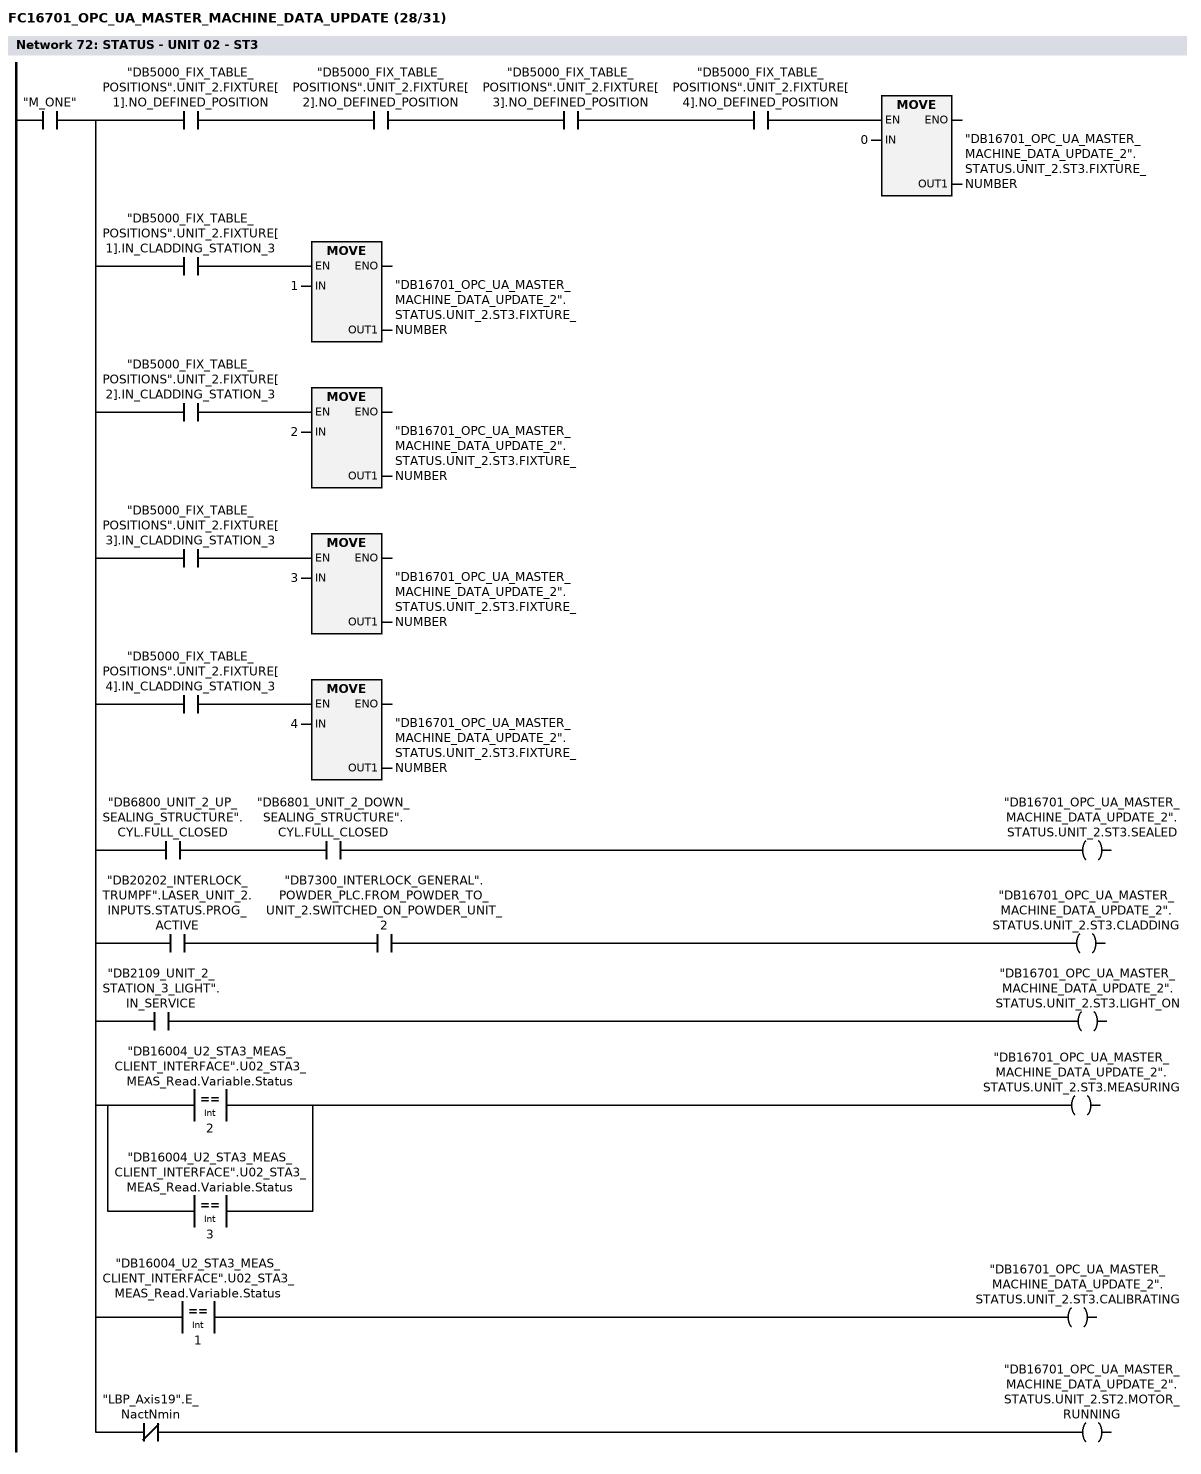
   RUNG wire#powerrail
      Contact( "M_ONE" )
      wire#w1
      Contact( "DB5000_FIX_TABLE_POSITIONS".UNIT_2.FIXTURE[1].NO_DEFINED_POSITION )
      Contact( "DB5000_FIX_TABLE_POSITIONS".UNIT_2.FIXTURE[2].NO_DEFINED_POSITION )
      Contact( "DB5000_FIX_TABLE_POSITIONS".UNIT_2.FIXTURE[3].NO_DEFINED_POSITION )
      Contact( "DB5000_FIX_TABLE_POSITIONS".UNIT_2.FIXTURE[4].NO_DEFINED_POSITION )
      Move(in := 0, out1 => "DB16701_OPC_UA_MASTER_MACHINE_DATA_UPDATE_2".STATUS.UNIT_2.ST3.FIXTURE_NUMBER)
   END_RUNG
   RUNG wire#w1
      Contact( "DB5000_FIX_TABLE_POSITIONS".UNIT_2.FIXTURE[1].IN_CLADDING_STATION_3 )
      Move(in := 1, out1 => "DB16701_OPC_UA_MASTER_MACHINE_DATA_UPDATE_2".STATUS.UNIT_2.ST3.FIXTURE_NUMBER)
   END_RUNG
   RUNG wire#w1
      Contact( "DB5000_FIX_TABLE_POSITIONS".UNIT_2.FIXTURE[2].IN_CLADDING_STATION_3 )
      Move(in := 2, out1 => "DB16701_OPC_UA_MASTER_MACHINE_DATA_UPDATE_2".STATUS.UNIT_2.ST3.FIXTURE_NUMBER)
   END_RUNG
   RUNG wire#w1
      Contact( "DB5000_FIX_TABLE_POSITIONS".UNIT_2.FIXTURE[3].IN_CLADDING_STATION_3 )
      Move(in := 3, out1 => "DB16701_OPC_UA_MASTER_MACHINE_DATA_UPDATE_2".STATUS.UNIT_2.ST3.FIXTURE_NUMBER)
   END_RUNG
   RUNG wire#w1
      Contact( "DB5000_FIX_TABLE_POSITIONS".UNIT_2.FIXTURE[4].IN_CLADDING_STATION_3 )
      Move(in := 4, out1 => "DB16701_OPC_UA_MASTER_MACHINE_DATA_UPDATE_2".STATUS.UNIT_2.ST3.FIXTURE_NUMBER)
   END_RUNG
   RUNG wire#w1
      Contact( "DB6800_UNIT_2_UP_SEALING_STRUCTURE".CYL.FULL_CLOSED )
      Contact( "DB6801_UNIT_2_DOWN_SEALING_STRUCTURE".CYL.FULL_CLOSED )
      Coil( "DB16701_OPC_UA_MASTER_MACHINE_DATA_UPDATE_2".STATUS.UNIT_2.ST3.SEALED )
   END_RUNG
   RUNG wire#w1
      Contact( "DB20202_INTERLOCK_TRUMPF".LASER_UNIT_2.INPUTS.STATUS.PROG_ACTIVE )
      Contact( "DB7300_INTERLOCK_GENERAL".POWDER_PLC.FROM_POWDER_TO_UNIT_2.SWITCHED_ON_POWDER_UNIT_2 )
      Coil( "DB16701_OPC_UA_MASTER_MACHINE_DATA_UPDATE_2".STATUS.UNIT_2.ST3.CLADDING )
   END_RUNG
   RUNG wire#w1
      Contact( "DB2109_UNIT_2_STATION_3_LIGHT".IN_SERVICE )
      Coil( "DB16701_OPC_UA_MASTER_MACHINE_DATA_UPDATE_2".STATUS.UNIT_2.ST3.LIGHT_ON )
   END_RUNG
   RUNG wire#w1
      { S7_Templates := "SrcType := Int" } EQ_Contact(in1 := "DB16004_U2_STA3_MEAS_CLIENT_INTERFACE".U02_STA3_MEAS_Read.Variable.Status, in2 := 2)
      wire#w2
      Coil( "DB16701_OPC_UA_MASTER_MACHINE_DATA_UPDATE_2".STATUS.UNIT_2.ST3.MEASURING )
   END_RUNG
   RUNG wire#w1
      { S7_Templates := "SrcType := Int" } EQ_Contact(in1 := "DB16004_U2_STA3_MEAS_CLIENT_INTERFACE".U02_STA3_MEAS_Read.Variable.Status, in2 := 3)
   END_RUNG wire#w2
   RUNG wire#w1
      { S7_Templates := "SrcType := Int" } EQ_Contact(in1 := "DB16004_U2_STA3_MEAS_CLIENT_INTERFACE".U02_STA3_MEAS_Read.Variable.Status, in2 := 1)
      Coil( "DB16701_OPC_UA_MASTER_MACHINE_DATA_UPDATE_2".STATUS.UNIT_2.ST3.CALIBRATING )
   END_RUNG
   RUNG wire#w1
      I_Contact( "LBP_Axis19".E_NactNmin )
      Coil( "DB16701_OPC_UA_MASTER_MACHINE_DATA_UPDATE_2".STATUS.UNIT_2.ST2.MOTOR_RUNNING )
   END_RUNG
   // the same network as SCL:
   IF "M_ONE" AND "DB5000_FIX_TABLE_POSITIONS".UNIT_2.FIXTURE[1].NO_DEFINED_POSITION AND "DB5000_FIX_TABLE_POSITIONS".UNIT_2.FIXTURE[2].NO_DEFINED_POSITION AND "DB5000_FIX_TABLE_POSITIONS".UNIT_2.FIXTURE[3].NO_DEFINED_POSITION AND "DB5000_FIX_TABLE_POSITIONS".UNIT_2.FIXTURE[4].NO_DEFINED_POSITION THEN
       "DB16701_OPC_UA_MASTER_MACHINE_DATA_UPDATE_2".STATUS.UNIT_2.ST3.FIXTURE_NUMBER := 0;
   END_IF;
   IF "M_ONE" AND "DB5000_FIX_TABLE_POSITIONS".UNIT_2.FIXTURE[1].IN_CLADDING_STATION_3 THEN
       "DB16701_OPC_UA_MASTER_MACHINE_DATA_UPDATE_2".STATUS.UNIT_2.ST3.FIXTURE_NUMBER := 1;
   END_IF;
   IF "M_ONE" AND "DB5000_FIX_TABLE_POSITIONS".UNIT_2.FIXTURE[2].IN_CLADDING_STATION_3 THEN
       "DB16701_OPC_UA_MASTER_MACHINE_DATA_UPDATE_2".STATUS.UNIT_2.ST3.FIXTURE_NUMBER := 2;
   END_IF;
   IF "M_ONE" AND "DB5000_FIX_TABLE_POSITIONS".UNIT_2.FIXTURE[3].IN_CLADDING_STATION_3 THEN
       "DB16701_OPC_UA_MASTER_MACHINE_DATA_UPDATE_2".STATUS.UNIT_2.ST3.FIXTURE_NUMBER := 3;
   END_IF;
   IF "M_ONE" AND "DB5000_FIX_TABLE_POSITIONS".UNIT_2.FIXTURE[4].IN_CLADDING_STATION_3 THEN
       "DB16701_OPC_UA_MASTER_MACHINE_DATA_UPDATE_2".STATUS.UNIT_2.ST3.FIXTURE_NUMBER := 4;
   END_IF;
   "DB16701_OPC_UA_MASTER_MACHINE_DATA_UPDATE_2".STATUS.UNIT_2.ST3.SEALED := "M_ONE" AND "DB6800_UNIT_2_UP_SEALING_STRUCTURE".CYL.FULL_CLOSED AND "DB6801_UNIT_2_DOWN_SEALING_STRUCTURE".CYL.FULL_CLOSED;
   "DB16701_OPC_UA_MASTER_MACHINE_DATA_UPDATE_2".STATUS.UNIT_2.ST3.CLADDING := "M_ONE" AND "DB20202_INTERLOCK_TRUMPF".LASER_UNIT_2.INPUTS.STATUS.PROG_ACTIVE AND "DB7300_INTERLOCK_GENERAL".POWDER_PLC.FROM_POWDER_TO_UNIT_2.SWITCHED_ON_POWDER_UNIT_2;
   "DB16701_OPC_UA_MASTER_MACHINE_DATA_UPDATE_2".STATUS.UNIT_2.ST3.LIGHT_ON := "M_ONE" AND "DB2109_UNIT_2_STATION_3_LIGHT".IN_SERVICE;
   "DB16701_OPC_UA_MASTER_MACHINE_DATA_UPDATE_2".STATUS.UNIT_2.ST3.MEASURING := "M_ONE" AND (("DB16004_U2_STA3_MEAS_CLIENT_INTERFACE".U02_STA3_MEAS_Read.Variable.Status = 2) OR ("DB16004_U2_STA3_MEAS_CLIENT_INTERFACE".U02_STA3_MEAS_Read.Variable.Status = 3));
   "DB16701_OPC_UA_MASTER_MACHINE_DATA_UPDATE_2".STATUS.UNIT_2.ST3.CALIBRATING := "M_ONE" AND ("DB16004_U2_STA3_MEAS_CLIENT_INTERFACE".U02_STA3_MEAS_Read.Variable.Status = 1);
   "DB16701_OPC_UA_MASTER_MACHINE_DATA_UPDATE_2".STATUS.UNIT_2.ST2.MOTOR_RUNNING := "M_ONE" AND NOT "LBP_Axis19".E_NactNmin;
END_REGION

REGION Network 73: STATUS - UNIT 02 - ST4
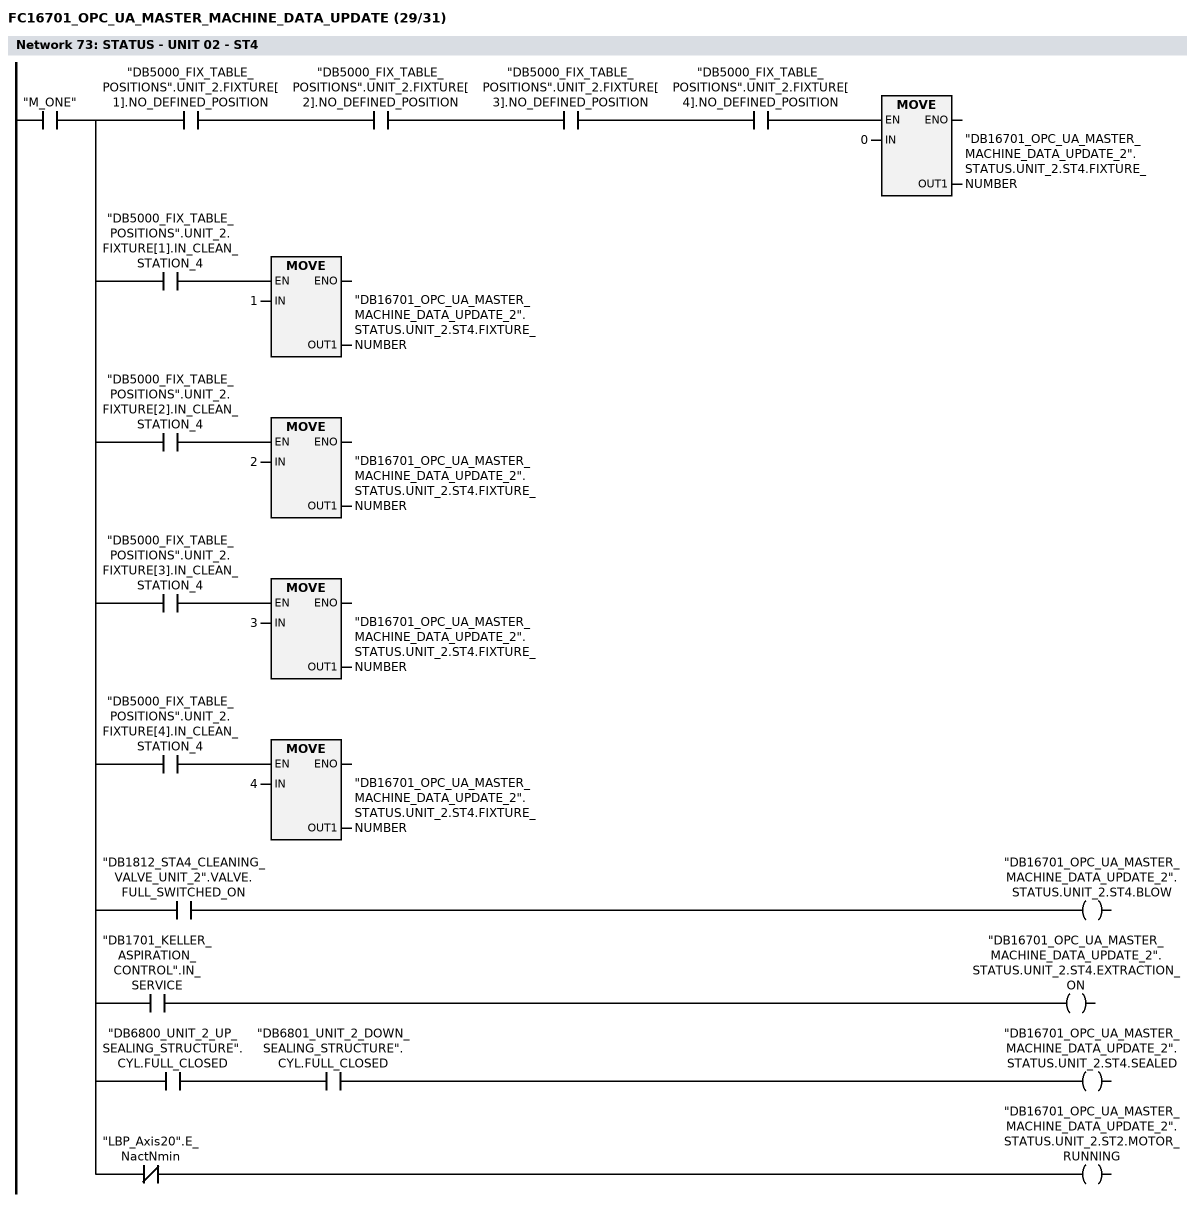
   RUNG wire#powerrail
      Contact( "M_ONE" )
      wire#w1
      Contact( "DB5000_FIX_TABLE_POSITIONS".UNIT_2.FIXTURE[1].NO_DEFINED_POSITION )
      Contact( "DB5000_FIX_TABLE_POSITIONS".UNIT_2.FIXTURE[2].NO_DEFINED_POSITION )
      Contact( "DB5000_FIX_TABLE_POSITIONS".UNIT_2.FIXTURE[3].NO_DEFINED_POSITION )
      Contact( "DB5000_FIX_TABLE_POSITIONS".UNIT_2.FIXTURE[4].NO_DEFINED_POSITION )
      Move(in := 0, out1 => "DB16701_OPC_UA_MASTER_MACHINE_DATA_UPDATE_2".STATUS.UNIT_2.ST4.FIXTURE_NUMBER)
   END_RUNG
   RUNG wire#w1
      Contact( "DB5000_FIX_TABLE_POSITIONS".UNIT_2.FIXTURE[1].IN_CLEAN_STATION_4 )
      Move(in := 1, out1 => "DB16701_OPC_UA_MASTER_MACHINE_DATA_UPDATE_2".STATUS.UNIT_2.ST4.FIXTURE_NUMBER)
   END_RUNG
   RUNG wire#w1
      Contact( "DB5000_FIX_TABLE_POSITIONS".UNIT_2.FIXTURE[2].IN_CLEAN_STATION_4 )
      Move(in := 2, out1 => "DB16701_OPC_UA_MASTER_MACHINE_DATA_UPDATE_2".STATUS.UNIT_2.ST4.FIXTURE_NUMBER)
   END_RUNG
   RUNG wire#w1
      Contact( "DB5000_FIX_TABLE_POSITIONS".UNIT_2.FIXTURE[3].IN_CLEAN_STATION_4 )
      Move(in := 3, out1 => "DB16701_OPC_UA_MASTER_MACHINE_DATA_UPDATE_2".STATUS.UNIT_2.ST4.FIXTURE_NUMBER)
   END_RUNG
   RUNG wire#w1
      Contact( "DB5000_FIX_TABLE_POSITIONS".UNIT_2.FIXTURE[4].IN_CLEAN_STATION_4 )
      Move(in := 4, out1 => "DB16701_OPC_UA_MASTER_MACHINE_DATA_UPDATE_2".STATUS.UNIT_2.ST4.FIXTURE_NUMBER)
   END_RUNG
   RUNG wire#w1
      Contact( "DB1812_STA4_CLEANING_VALVE_UNIT_2".VALVE.FULL_SWITCHED_ON )
      Coil( "DB16701_OPC_UA_MASTER_MACHINE_DATA_UPDATE_2".STATUS.UNIT_2.ST4.BLOW )
   END_RUNG
   RUNG wire#w1
      Contact( "DB1701_KELLER_ASPIRATION_CONTROL".IN_SERVICE )
      Coil( "DB16701_OPC_UA_MASTER_MACHINE_DATA_UPDATE_2".STATUS.UNIT_2.ST4.EXTRACTION_ON )
   END_RUNG
   RUNG wire#w1
      Contact( "DB6800_UNIT_2_UP_SEALING_STRUCTURE".CYL.FULL_CLOSED )
      Contact( "DB6801_UNIT_2_DOWN_SEALING_STRUCTURE".CYL.FULL_CLOSED )
      Coil( "DB16701_OPC_UA_MASTER_MACHINE_DATA_UPDATE_2".STATUS.UNIT_2.ST4.SEALED )
   END_RUNG
   RUNG wire#w1
      I_Contact( "LBP_Axis20".E_NactNmin )
      Coil( "DB16701_OPC_UA_MASTER_MACHINE_DATA_UPDATE_2".STATUS.UNIT_2.ST2.MOTOR_RUNNING )
   END_RUNG
   // the same network as SCL:
   IF "M_ONE" AND "DB5000_FIX_TABLE_POSITIONS".UNIT_2.FIXTURE[1].NO_DEFINED_POSITION AND "DB5000_FIX_TABLE_POSITIONS".UNIT_2.FIXTURE[2].NO_DEFINED_POSITION AND "DB5000_FIX_TABLE_POSITIONS".UNIT_2.FIXTURE[3].NO_DEFINED_POSITION AND "DB5000_FIX_TABLE_POSITIONS".UNIT_2.FIXTURE[4].NO_DEFINED_POSITION THEN
       "DB16701_OPC_UA_MASTER_MACHINE_DATA_UPDATE_2".STATUS.UNIT_2.ST4.FIXTURE_NUMBER := 0;
   END_IF;
   IF "M_ONE" AND "DB5000_FIX_TABLE_POSITIONS".UNIT_2.FIXTURE[1].IN_CLEAN_STATION_4 THEN
       "DB16701_OPC_UA_MASTER_MACHINE_DATA_UPDATE_2".STATUS.UNIT_2.ST4.FIXTURE_NUMBER := 1;
   END_IF;
   IF "M_ONE" AND "DB5000_FIX_TABLE_POSITIONS".UNIT_2.FIXTURE[2].IN_CLEAN_STATION_4 THEN
       "DB16701_OPC_UA_MASTER_MACHINE_DATA_UPDATE_2".STATUS.UNIT_2.ST4.FIXTURE_NUMBER := 2;
   END_IF;
   IF "M_ONE" AND "DB5000_FIX_TABLE_POSITIONS".UNIT_2.FIXTURE[3].IN_CLEAN_STATION_4 THEN
       "DB16701_OPC_UA_MASTER_MACHINE_DATA_UPDATE_2".STATUS.UNIT_2.ST4.FIXTURE_NUMBER := 3;
   END_IF;
   IF "M_ONE" AND "DB5000_FIX_TABLE_POSITIONS".UNIT_2.FIXTURE[4].IN_CLEAN_STATION_4 THEN
       "DB16701_OPC_UA_MASTER_MACHINE_DATA_UPDATE_2".STATUS.UNIT_2.ST4.FIXTURE_NUMBER := 4;
   END_IF;
   "DB16701_OPC_UA_MASTER_MACHINE_DATA_UPDATE_2".STATUS.UNIT_2.ST4.BLOW := "M_ONE" AND "DB1812_STA4_CLEANING_VALVE_UNIT_2".VALVE.FULL_SWITCHED_ON;
   "DB16701_OPC_UA_MASTER_MACHINE_DATA_UPDATE_2".STATUS.UNIT_2.ST4.EXTRACTION_ON := "M_ONE" AND "DB1701_KELLER_ASPIRATION_CONTROL".IN_SERVICE;
   "DB16701_OPC_UA_MASTER_MACHINE_DATA_UPDATE_2".STATUS.UNIT_2.ST4.SEALED := "M_ONE" AND "DB6800_UNIT_2_UP_SEALING_STRUCTURE".CYL.FULL_CLOSED AND "DB6801_UNIT_2_DOWN_SEALING_STRUCTURE".CYL.FULL_CLOSED;
   "DB16701_OPC_UA_MASTER_MACHINE_DATA_UPDATE_2".STATUS.UNIT_2.ST2.MOTOR_RUNNING := "M_ONE" AND NOT "LBP_Axis20".E_NactNmin;
END_REGION

REGION Network 74: STATUS - UNIT 02 - F1
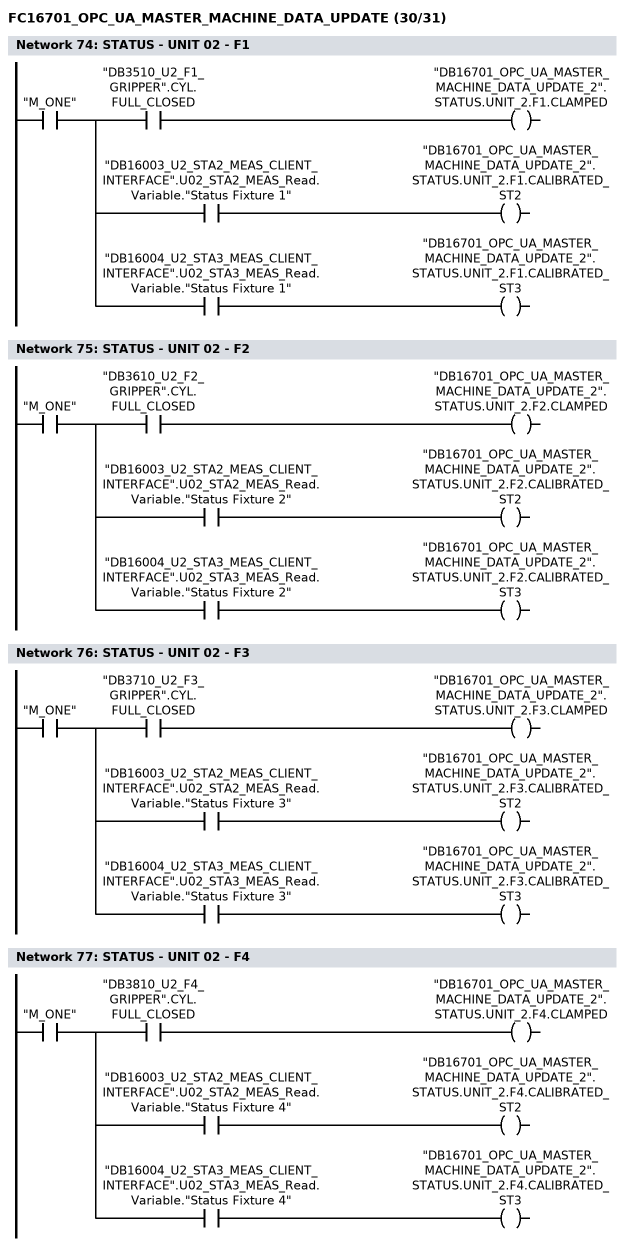
   RUNG wire#powerrail
      Contact( "M_ONE" )
      wire#w1
      Contact( "DB3510_U2_F1_GRIPPER".CYL.FULL_CLOSED )
      Coil( "DB16701_OPC_UA_MASTER_MACHINE_DATA_UPDATE_2".STATUS.UNIT_2.F1.CLAMPED )
   END_RUNG
   RUNG wire#w1
      Contact( "DB16003_U2_STA2_MEAS_CLIENT_INTERFACE".U02_STA2_MEAS_Read.Variable."Status Fixture 1" )
      Coil( "DB16701_OPC_UA_MASTER_MACHINE_DATA_UPDATE_2".STATUS.UNIT_2.F1.CALIBRATED_ST2 )
   END_RUNG
   RUNG wire#w1
      Contact( "DB16004_U2_STA3_MEAS_CLIENT_INTERFACE".U02_STA3_MEAS_Read.Variable."Status Fixture 1" )
      Coil( "DB16701_OPC_UA_MASTER_MACHINE_DATA_UPDATE_2".STATUS.UNIT_2.F1.CALIBRATED_ST3 )
   END_RUNG
   // the same network as SCL:
   "DB16701_OPC_UA_MASTER_MACHINE_DATA_UPDATE_2".STATUS.UNIT_2.F1.CLAMPED := "M_ONE" AND "DB3510_U2_F1_GRIPPER".CYL.FULL_CLOSED;
   "DB16701_OPC_UA_MASTER_MACHINE_DATA_UPDATE_2".STATUS.UNIT_2.F1.CALIBRATED_ST2 := "M_ONE" AND "DB16003_U2_STA2_MEAS_CLIENT_INTERFACE".U02_STA2_MEAS_Read.Variable."Status Fixture 1";
   "DB16701_OPC_UA_MASTER_MACHINE_DATA_UPDATE_2".STATUS.UNIT_2.F1.CALIBRATED_ST3 := "M_ONE" AND "DB16004_U2_STA3_MEAS_CLIENT_INTERFACE".U02_STA3_MEAS_Read.Variable."Status Fixture 1";
END_REGION

REGION Network 75: STATUS - UNIT 02 - F2
   RUNG wire#powerrail
      Contact( "M_ONE" )
      wire#w1
      Contact( "DB3610_U2_F2_GRIPPER".CYL.FULL_CLOSED )
      Coil( "DB16701_OPC_UA_MASTER_MACHINE_DATA_UPDATE_2".STATUS.UNIT_2.F2.CLAMPED )
   END_RUNG
   RUNG wire#w1
      Contact( "DB16003_U2_STA2_MEAS_CLIENT_INTERFACE".U02_STA2_MEAS_Read.Variable."Status Fixture 2" )
      Coil( "DB16701_OPC_UA_MASTER_MACHINE_DATA_UPDATE_2".STATUS.UNIT_2.F2.CALIBRATED_ST2 )
   END_RUNG
   RUNG wire#w1
      Contact( "DB16004_U2_STA3_MEAS_CLIENT_INTERFACE".U02_STA3_MEAS_Read.Variable."Status Fixture 2" )
      Coil( "DB16701_OPC_UA_MASTER_MACHINE_DATA_UPDATE_2".STATUS.UNIT_2.F2.CALIBRATED_ST3 )
   END_RUNG
   // the same network as SCL:
   "DB16701_OPC_UA_MASTER_MACHINE_DATA_UPDATE_2".STATUS.UNIT_2.F2.CLAMPED := "M_ONE" AND "DB3610_U2_F2_GRIPPER".CYL.FULL_CLOSED;
   "DB16701_OPC_UA_MASTER_MACHINE_DATA_UPDATE_2".STATUS.UNIT_2.F2.CALIBRATED_ST2 := "M_ONE" AND "DB16003_U2_STA2_MEAS_CLIENT_INTERFACE".U02_STA2_MEAS_Read.Variable."Status Fixture 2";
   "DB16701_OPC_UA_MASTER_MACHINE_DATA_UPDATE_2".STATUS.UNIT_2.F2.CALIBRATED_ST3 := "M_ONE" AND "DB16004_U2_STA3_MEAS_CLIENT_INTERFACE".U02_STA3_MEAS_Read.Variable."Status Fixture 2";
END_REGION

REGION Network 76: STATUS - UNIT 02 - F3
   RUNG wire#powerrail
      Contact( "M_ONE" )
      wire#w1
      Contact( "DB3710_U2_F3_GRIPPER".CYL.FULL_CLOSED )
      Coil( "DB16701_OPC_UA_MASTER_MACHINE_DATA_UPDATE_2".STATUS.UNIT_2.F3.CLAMPED )
   END_RUNG
   RUNG wire#w1
      Contact( "DB16003_U2_STA2_MEAS_CLIENT_INTERFACE".U02_STA2_MEAS_Read.Variable."Status Fixture 3" )
      Coil( "DB16701_OPC_UA_MASTER_MACHINE_DATA_UPDATE_2".STATUS.UNIT_2.F3.CALIBRATED_ST2 )
   END_RUNG
   RUNG wire#w1
      Contact( "DB16004_U2_STA3_MEAS_CLIENT_INTERFACE".U02_STA3_MEAS_Read.Variable."Status Fixture 3" )
      Coil( "DB16701_OPC_UA_MASTER_MACHINE_DATA_UPDATE_2".STATUS.UNIT_2.F3.CALIBRATED_ST3 )
   END_RUNG
   // the same network as SCL:
   "DB16701_OPC_UA_MASTER_MACHINE_DATA_UPDATE_2".STATUS.UNIT_2.F3.CLAMPED := "M_ONE" AND "DB3710_U2_F3_GRIPPER".CYL.FULL_CLOSED;
   "DB16701_OPC_UA_MASTER_MACHINE_DATA_UPDATE_2".STATUS.UNIT_2.F3.CALIBRATED_ST2 := "M_ONE" AND "DB16003_U2_STA2_MEAS_CLIENT_INTERFACE".U02_STA2_MEAS_Read.Variable."Status Fixture 3";
   "DB16701_OPC_UA_MASTER_MACHINE_DATA_UPDATE_2".STATUS.UNIT_2.F3.CALIBRATED_ST3 := "M_ONE" AND "DB16004_U2_STA3_MEAS_CLIENT_INTERFACE".U02_STA3_MEAS_Read.Variable."Status Fixture 3";
END_REGION

REGION Network 77: STATUS - UNIT 02 - F4
   RUNG wire#powerrail
      Contact( "M_ONE" )
      wire#w1
      Contact( "DB3810_U2_F4_GRIPPER".CYL.FULL_CLOSED )
      Coil( "DB16701_OPC_UA_MASTER_MACHINE_DATA_UPDATE_2".STATUS.UNIT_2.F4.CLAMPED )
   END_RUNG
   RUNG wire#w1
      Contact( "DB16003_U2_STA2_MEAS_CLIENT_INTERFACE".U02_STA2_MEAS_Read.Variable."Status Fixture 4" )
      Coil( "DB16701_OPC_UA_MASTER_MACHINE_DATA_UPDATE_2".STATUS.UNIT_2.F4.CALIBRATED_ST2 )
   END_RUNG
   RUNG wire#w1
      Contact( "DB16004_U2_STA3_MEAS_CLIENT_INTERFACE".U02_STA3_MEAS_Read.Variable."Status Fixture 4" )
      Coil( "DB16701_OPC_UA_MASTER_MACHINE_DATA_UPDATE_2".STATUS.UNIT_2.F4.CALIBRATED_ST3 )
   END_RUNG
   // the same network as SCL:
   "DB16701_OPC_UA_MASTER_MACHINE_DATA_UPDATE_2".STATUS.UNIT_2.F4.CLAMPED := "M_ONE" AND "DB3810_U2_F4_GRIPPER".CYL.FULL_CLOSED;
   "DB16701_OPC_UA_MASTER_MACHINE_DATA_UPDATE_2".STATUS.UNIT_2.F4.CALIBRATED_ST2 := "M_ONE" AND "DB16003_U2_STA2_MEAS_CLIENT_INTERFACE".U02_STA2_MEAS_Read.Variable."Status Fixture 4";
   "DB16701_OPC_UA_MASTER_MACHINE_DATA_UPDATE_2".STATUS.UNIT_2.F4.CALIBRATED_ST3 := "M_ONE" AND "DB16004_U2_STA3_MEAS_CLIENT_INTERFACE".U02_STA3_MEAS_Read.Variable."Status Fixture 4";
END_REGION

REGION Network 78: STATUS - UNIT 02 - LASER
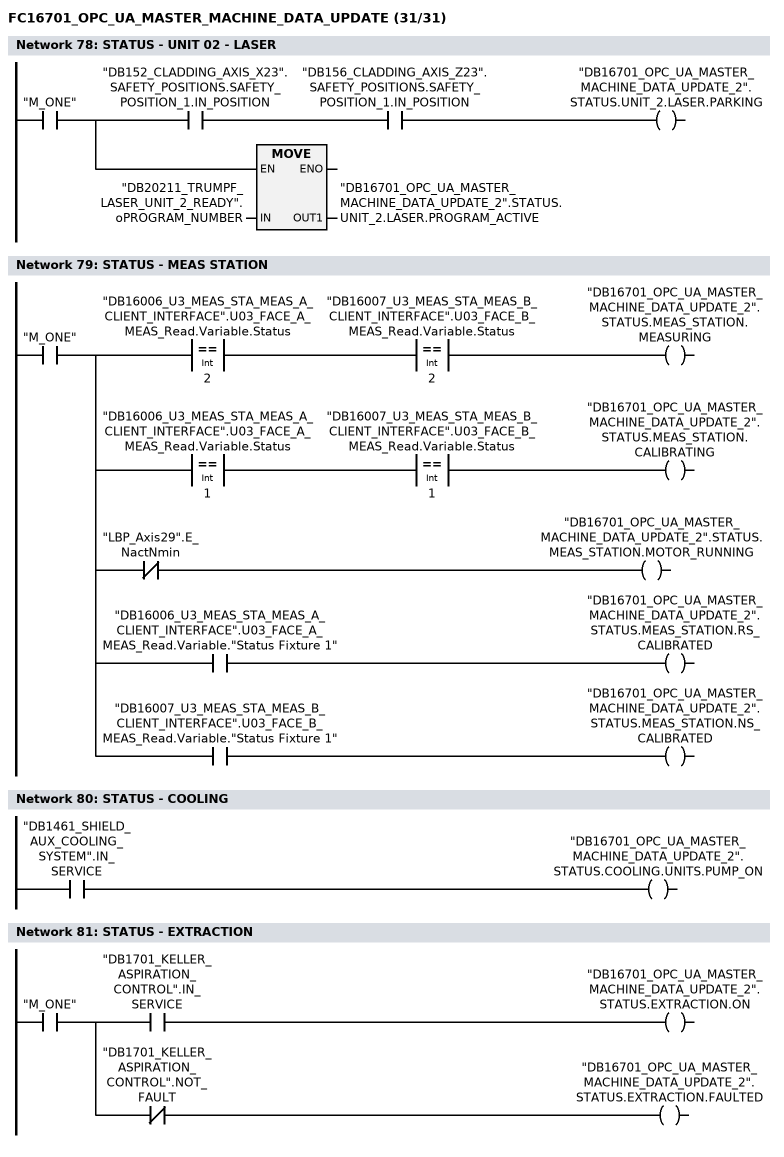
   RUNG wire#powerrail
      Contact( "M_ONE" )
      wire#w1
      Contact( "DB152_CLADDING_AXIS_X23".SAFETY_POSITIONS.SAFETY_POSITION_1.IN_POSITION )
      Contact( "DB156_CLADDING_AXIS_Z23".SAFETY_POSITIONS.SAFETY_POSITION_1.IN_POSITION )
      Coil( "DB16701_OPC_UA_MASTER_MACHINE_DATA_UPDATE_2".STATUS.UNIT_2.LASER.PARKING )
   END_RUNG
   RUNG wire#w1
      Move(in := "DB20211_TRUMPF_LASER_UNIT_2_READY".oPROGRAM_NUMBER, out1 => "DB16701_OPC_UA_MASTER_MACHINE_DATA_UPDATE_2".STATUS.UNIT_2.LASER.PROGRAM_ACTIVE)
   END_RUNG
   // the same network as SCL:
   "DB16701_OPC_UA_MASTER_MACHINE_DATA_UPDATE_2".STATUS.UNIT_2.LASER.PARKING := "M_ONE" AND "DB152_CLADDING_AXIS_X23".SAFETY_POSITIONS.SAFETY_POSITION_1.IN_POSITION AND "DB156_CLADDING_AXIS_Z23".SAFETY_POSITIONS.SAFETY_POSITION_1.IN_POSITION;
   IF "M_ONE" THEN
       "DB16701_OPC_UA_MASTER_MACHINE_DATA_UPDATE_2".STATUS.UNIT_2.LASER.PROGRAM_ACTIVE := "DB20211_TRUMPF_LASER_UNIT_2_READY".oPROGRAM_NUMBER;
   END_IF;
END_REGION

REGION Network 79: STATUS - MEAS STATION
   RUNG wire#powerrail
      Contact( "M_ONE" )
      wire#w1
      { S7_Templates := "SrcType := Int" } EQ_Contact(in1 := "DB16006_U3_MEAS_STA_MEAS_A_CLIENT_INTERFACE".U03_FACE_A_MEAS_Read.Variable.Status, in2 := 2)
      { S7_Templates := "SrcType := Int" } EQ_Contact(in1 := "DB16007_U3_MEAS_STA_MEAS_B_CLIENT_INTERFACE".U03_FACE_B_MEAS_Read.Variable.Status, in2 := 2)
      Coil( "DB16701_OPC_UA_MASTER_MACHINE_DATA_UPDATE_2".STATUS.MEAS_STATION.MEASURING )
   END_RUNG
   RUNG wire#w1
      { S7_Templates := "SrcType := Int" } EQ_Contact(in1 := "DB16006_U3_MEAS_STA_MEAS_A_CLIENT_INTERFACE".U03_FACE_A_MEAS_Read.Variable.Status, in2 := 1)
      { S7_Templates := "SrcType := Int" } EQ_Contact(in1 := "DB16007_U3_MEAS_STA_MEAS_B_CLIENT_INTERFACE".U03_FACE_B_MEAS_Read.Variable.Status, in2 := 1)
      Coil( "DB16701_OPC_UA_MASTER_MACHINE_DATA_UPDATE_2".STATUS.MEAS_STATION.CALIBRATING )
   END_RUNG
   RUNG wire#w1
      I_Contact( "LBP_Axis29".E_NactNmin )
      Coil( "DB16701_OPC_UA_MASTER_MACHINE_DATA_UPDATE_2".STATUS.MEAS_STATION.MOTOR_RUNNING )
   END_RUNG
   RUNG wire#w1
      Contact( "DB16006_U3_MEAS_STA_MEAS_A_CLIENT_INTERFACE".U03_FACE_A_MEAS_Read.Variable."Status Fixture 1" )
      Coil( "DB16701_OPC_UA_MASTER_MACHINE_DATA_UPDATE_2".STATUS.MEAS_STATION.RS_CALIBRATED )
   END_RUNG
   RUNG wire#w1
      Contact( "DB16007_U3_MEAS_STA_MEAS_B_CLIENT_INTERFACE".U03_FACE_B_MEAS_Read.Variable."Status Fixture 1" )
      Coil( "DB16701_OPC_UA_MASTER_MACHINE_DATA_UPDATE_2".STATUS.MEAS_STATION.NS_CALIBRATED )
   END_RUNG
   // the same network as SCL:
   "DB16701_OPC_UA_MASTER_MACHINE_DATA_UPDATE_2".STATUS.MEAS_STATION.MEASURING := "M_ONE" AND ("DB16006_U3_MEAS_STA_MEAS_A_CLIENT_INTERFACE".U03_FACE_A_MEAS_Read.Variable.Status = 2) AND ("DB16007_U3_MEAS_STA_MEAS_B_CLIENT_INTERFACE".U03_FACE_B_MEAS_Read.Variable.Status = 2);
   "DB16701_OPC_UA_MASTER_MACHINE_DATA_UPDATE_2".STATUS.MEAS_STATION.CALIBRATING := "M_ONE" AND ("DB16006_U3_MEAS_STA_MEAS_A_CLIENT_INTERFACE".U03_FACE_A_MEAS_Read.Variable.Status = 1) AND ("DB16007_U3_MEAS_STA_MEAS_B_CLIENT_INTERFACE".U03_FACE_B_MEAS_Read.Variable.Status = 1);
   "DB16701_OPC_UA_MASTER_MACHINE_DATA_UPDATE_2".STATUS.MEAS_STATION.MOTOR_RUNNING := "M_ONE" AND NOT "LBP_Axis29".E_NactNmin;
   "DB16701_OPC_UA_MASTER_MACHINE_DATA_UPDATE_2".STATUS.MEAS_STATION.RS_CALIBRATED := "M_ONE" AND "DB16006_U3_MEAS_STA_MEAS_A_CLIENT_INTERFACE".U03_FACE_A_MEAS_Read.Variable."Status Fixture 1";
   "DB16701_OPC_UA_MASTER_MACHINE_DATA_UPDATE_2".STATUS.MEAS_STATION.NS_CALIBRATED := "M_ONE" AND "DB16007_U3_MEAS_STA_MEAS_B_CLIENT_INTERFACE".U03_FACE_B_MEAS_Read.Variable."Status Fixture 1";
END_REGION

REGION Network 80: STATUS - COOLING
   RUNG wire#powerrail
      Contact( "DB1461_SHIELD_AUX_COOLING_SYSTEM".IN_SERVICE )
      Coil( "DB16701_OPC_UA_MASTER_MACHINE_DATA_UPDATE_2".STATUS.COOLING.UNITS.PUMP_ON )
   END_RUNG
   // the same network as SCL:
   "DB16701_OPC_UA_MASTER_MACHINE_DATA_UPDATE_2".STATUS.COOLING.UNITS.PUMP_ON := "DB1461_SHIELD_AUX_COOLING_SYSTEM".IN_SERVICE;
END_REGION

REGION Network 81: STATUS - EXTRACTION
   RUNG wire#powerrail
      Contact( "M_ONE" )
      wire#w1
      Contact( "DB1701_KELLER_ASPIRATION_CONTROL".IN_SERVICE )
      Coil( "DB16701_OPC_UA_MASTER_MACHINE_DATA_UPDATE_2".STATUS.EXTRACTION.ON )
   END_RUNG
   RUNG wire#w1
      I_Contact( "DB1701_KELLER_ASPIRATION_CONTROL".NOT_FAULT )
      Coil( "DB16701_OPC_UA_MASTER_MACHINE_DATA_UPDATE_2".STATUS.EXTRACTION.FAULTED )
   END_RUNG
   // the same network as SCL:
   "DB16701_OPC_UA_MASTER_MACHINE_DATA_UPDATE_2".STATUS.EXTRACTION.ON := "M_ONE" AND "DB1701_KELLER_ASPIRATION_CONTROL".IN_SERVICE;
   "DB16701_OPC_UA_MASTER_MACHINE_DATA_UPDATE_2".STATUS.EXTRACTION.FAULTED := "M_ONE" AND NOT "DB1701_KELLER_ASPIRATION_CONTROL".NOT_FAULT;
END_REGION

REGION Network 82: STATUS - MAINTENANCE---------------------------------------------------------
END_REGION
END_FUNCTION
